ACTION ACT_Move:
{region "Primary"}
mcMoveAbsolute(	Axis					:= Axis,
				Execute					:= stMcAxisOnline.mcMoveAbsolute.bExecute,
				Position				:= stMcAxisOnline.mcMoveAbsolute.lrPosition,
				Velocity				:= stMcAxisOnline.mcMoveAbsolute.lrVelocity,
				Acceleration			:= stMcAxisOnline.mcMoveAbsolute.lrAcceleration,
				Deceleration			:= stMcAxisOnline.mcMoveAbsolute.lrDeceleration,
				Jerk					:= stMcAxisOnline.mcMoveAbsolute.lrJerk,
				BufferMode				:= stMcAxisOnline.mcMoveAbsolute.eBufferMode,
				Options					:= stMcAxisOnline.mcMoveAbsolute.stOptions,
				Done					=> stMcAxisOnline.mcMoveAbsolute.bDone,
				Busy					=> stMcAxisOnline.mcMoveAbsolute.bBusy,
				Active					=> stMcAxisOnline.mcMoveAbsolute.bActive,
				CommandAborted			=> stMcAxisOnline.mcMoveAbsolute.bCommandAborted,
				Error					=> stMcAxisOnline.mcMoveAbsolute.bError,
				ErrorID					=> stMcAxisOnline.mcMoveAbsolute.udiErrorID);

mcMoveRelative(	Axis					:= Axis,
				Execute					:= stMcAxisOnline.mcMoveRelative.bExecute,
				Distance				:= stMcAxisOnline.mcMoveRelative.lrDistance,
				Velocity				:= stMcAxisOnline.mcMoveRelative.lrVelocity,
				Acceleration			:= stMcAxisOnline.mcMoveRelative.lrAcceleration,
				Deceleration			:= stMcAxisOnline.mcMoveRelative.lrDeceleration,
				Jerk					:= stMcAxisOnline.mcMoveRelative.lrJerk,
				BufferMode				:= stMcAxisOnline.mcMoveRelative.eBufferMode,
				Options					:= stMcAxisOnline.mcMoveRelative.stOptions,
				Done					=> stMcAxisOnline.mcMoveRelative.bDone,
				Busy					=> stMcAxisOnline.mcMoveRelative.bBusy,
				Active					=> stMcAxisOnline.mcMoveRelative.bActive,
				CommandAborted			=> stMcAxisOnline.mcMoveRelative.bCommandAborted,
				Error					=> stMcAxisOnline.mcMoveRelative.bError,
				ErrorID					=> stMcAxisOnline.mcMoveRelative.udiErrorID);
				
mcMoveVelocity(	Axis					:= Axis,
				Execute					:= stMcAxisOnline.mcMoveVelocity.bExecute,
				Velocity				:= stMcAxisOnline.mcMoveVelocity.lrVelocity,
				Acceleration			:= stMcAxisOnline.mcMoveVelocity.lrAcceleration,
				Deceleration			:= stMcAxisOnline.mcMoveVelocity.lrDeceleration,
				Jerk					:= stMcAxisOnline.mcMoveVelocity.lrJerk,
				Direction				:= stMcAxisOnline.mcMoveVelocity.eDirection,
				BufferMode				:= stMcAxisOnline.mcMoveVelocity.eBufferMode,
				Options					:= stMcAxisOnline.mcMoveVelocity.stOptions,
				InVelocity				=> stMcAxisOnline.mcMoveVelocity.bInVelocity,
				Busy					=> stMcAxisOnline.mcMoveVelocity.bBusy,
				Active					=> stMcAxisOnline.mcMoveVelocity.bActive,
				CommandAborted			=> stMcAxisOnline.mcMoveVelocity.bCommandAborted,
				Error					=> stMcAxisOnline.mcMoveVelocity.bError,
				ErrorID					=> stMcAxisOnline.mcMoveVelocity.udiErrorID);
stMcAxisOnline.mcMoveVelocity.bDone		:= stMcAxisOnline.mcMoveVelocity.bInVelocity;

mcMoveModulo(	Axis					:= Axis,
				Execute					:= stMcAxisOnline.mcMoveModulo.bExecute,
				Position				:= stMcAxisOnline.mcMoveModulo.lrPosition,
				Velocity				:= stMcAxisOnline.mcMoveModulo.lrVelocity,
				Acceleration			:= stMcAxisOnline.mcMoveModulo.lrAcceleration,
				Deceleration			:= stMcAxisOnline.mcMoveModulo.lrDeceleration,
				Jerk					:= stMcAxisOnline.mcMoveModulo.lrJerk,
				Direction				:= stMcAxisOnline.mcMoveModulo.eDirection,
				BufferMode				:= stMcAxisOnline.mcMoveModulo.eBufferMode,
				Options					:= stMcAxisOnline.mcMoveModulo.stOptions,
				Done					=> stMcAxisOnline.mcMoveModulo.bDone,
				Busy					=> stMcAxisOnline.mcMoveModulo.bBusy,
				Active					=> stMcAxisOnline.mcMoveModulo.bActive,
				CommandAborted			=> stMcAxisOnline.mcMoveModulo.bCommandAborted,
				Error					=> stMcAxisOnline.mcMoveModulo.bError,
				ErrorID					=> stMcAxisOnline.mcMoveModulo.udiErrorID);
{endregion}
{region "Secondary"}
mcMoveAbsolute2(Axis					:= Axis,
				Execute					:= stMcAxisOnline.mcMoveAbsolute2.bExecute,
				Position				:= stMcAxisOnline.mcMoveAbsolute2.lrPosition,
				Velocity				:= stMcAxisOnline.mcMoveAbsolute2.lrVelocity,
				Acceleration			:= stMcAxisOnline.mcMoveAbsolute2.lrAcceleration,
				Deceleration			:= stMcAxisOnline.mcMoveAbsolute2.lrDeceleration,
				Jerk					:= stMcAxisOnline.mcMoveAbsolute2.lrJerk,
				BufferMode				:= stMcAxisOnline.mcMoveAbsolute2.eBufferMode,
				Options					:= stMcAxisOnline.mcMoveAbsolute2.stOptions,
				Done					=> stMcAxisOnline.mcMoveAbsolute2.bDone,
				Busy					=> stMcAxisOnline.mcMoveAbsolute2.bBusy,
				Active					=> stMcAxisOnline.mcMoveAbsolute2.bActive,
				CommandAborted			=> stMcAxisOnline.mcMoveAbsolute2.bCommandAborted,
				Error					=> stMcAxisOnline.mcMoveAbsolute2.bError,
				ErrorID					=> stMcAxisOnline.mcMoveAbsolute2.udiErrorID);

mcMoveRelative2(Axis					:= Axis,
				Execute					:= stMcAxisOnline.mcMoveRelative2.bExecute,
				Distance				:= stMcAxisOnline.mcMoveRelative2.lrDistance,
				Velocity				:= stMcAxisOnline.mcMoveRelative2.lrVelocity,
				Acceleration			:= stMcAxisOnline.mcMoveRelative2.lrAcceleration,
				Deceleration			:= stMcAxisOnline.mcMoveRelative2.lrDeceleration,
				Jerk					:= stMcAxisOnline.mcMoveRelative2.lrJerk,
				BufferMode				:= stMcAxisOnline.mcMoveRelative2.eBufferMode,
				Options					:= stMcAxisOnline.mcMoveRelative2.stOptions,
				Done					=> stMcAxisOnline.mcMoveRelative2.bDone,
				Busy					=> stMcAxisOnline.mcMoveRelative2.bBusy,
				Active					=> stMcAxisOnline.mcMoveRelative2.bActive,
				CommandAborted			=> stMcAxisOnline.mcMoveRelative2.bCommandAborted,
				Error					=> stMcAxisOnline.mcMoveRelative2.bError,
				ErrorID					=> stMcAxisOnline.mcMoveRelative2.udiErrorID);
				
mcMoveVelocity2(Axis					:= Axis,
				Execute					:= stMcAxisOnline.mcMoveVelocity2.bExecute,
				Velocity				:= stMcAxisOnline.mcMoveVelocity2.lrVelocity,
				Acceleration			:= stMcAxisOnline.mcMoveVelocity2.lrAcceleration,
				Deceleration			:= stMcAxisOnline.mcMoveVelocity2.lrDeceleration,
				Jerk					:= stMcAxisOnline.mcMoveVelocity2.lrJerk,
				Direction				:= stMcAxisOnline.mcMoveVelocity2.eDirection,
				BufferMode				:= stMcAxisOnline.mcMoveVelocity2.eBufferMode,
				Options					:= stMcAxisOnline.mcMoveVelocity2.stOptions,
				InVelocity				=> stMcAxisOnline.mcMoveVelocity2.bInVelocity,
				Busy					=> stMcAxisOnline.mcMoveVelocity2.bBusy,
				Active					=> stMcAxisOnline.mcMoveVelocity2.bActive,
				CommandAborted			=> stMcAxisOnline.mcMoveVelocity2.bCommandAborted,
				Error					=> stMcAxisOnline.mcMoveVelocity2.bError,
				ErrorID					=> stMcAxisOnline.mcMoveVelocity2.udiErrorID);
stMcAxisOnline.mcMoveVelocity2.bDone	:= stMcAxisOnline.mcMoveVelocity2.bInVelocity;

mcMoveModulo2(	Axis					:= Axis,
				Execute					:= stMcAxisOnline.mcMoveModulo2.bExecute,
				Position				:= stMcAxisOnline.mcMoveModulo2.lrPosition,
				Velocity				:= stMcAxisOnline.mcMoveModulo2.lrVelocity,
				Acceleration			:= stMcAxisOnline.mcMoveModulo2.lrAcceleration,
				Deceleration			:= stMcAxisOnline.mcMoveModulo2.lrDeceleration,
				Jerk					:= stMcAxisOnline.mcMoveModulo2.lrJerk,
				Direction				:= stMcAxisOnline.mcMoveModulo2.eDirection,
				BufferMode				:= stMcAxisOnline.mcMoveModulo2.eBufferMode,
				Options					:= stMcAxisOnline.mcMoveModulo2.stOptions,
				Done					=> stMcAxisOnline.mcMoveModulo2.bDone,
				Busy					=> stMcAxisOnline.mcMoveModulo2.bBusy,
				Active					=> stMcAxisOnline.mcMoveModulo2.bActive,
				CommandAborted			=> stMcAxisOnline.mcMoveModulo2.bCommandAborted,
				Error					=> stMcAxisOnline.mcMoveModulo2.bError,
				ErrorID					=> stMcAxisOnline.mcMoveModulo2.udiErrorID);
{endregion}
END_ACTION

ACTION ACT_Power:
mcPower(	Axis						:= Axis,									//
			Enable						:= stMcAxisOnline.mcPower.bEnable,
			Enable_Positive				:= stMcAxisOnline.mcPower.bEnable_Positive,
			Enable_Negative				:= stMcAxisOnline.mcPower.bEnable_Negative,
			Override					:= stMcAxisOnline.mcPower.lrOverride,
			BufferMode					:= stMcAxisOnline.mcPower.eBufferMode,
			Options						:= stMcAxisOnline.mcPower.stOptions,
			Status						=> stMcAxisOnline.mcPower.bStatus,
			Busy						=> stMcAxisOnline.mcPower.bBusy,
			Active						=> stMcAxisOnline.mcPower.bActive,
			Error						=> stMcAxisOnline.mcPower.bError,
			ErrorID						=> stMcAxisOnline.mcPower.udiErrorID);
END_ACTION

ACTION ACT_ResetAndDiag:
tonGetDriveDiag(IN:= stMcAxisOnline.stError.bDriveError AND NOT tonGetDriveDiag.Q, PT:= T#5S, Q=> , ET=> );

IF Axis.Status.OpMode.SimulationAxis THEN
	mcReset(
		Axis						:= Axis,
		Execute						:= stMcAxisOnline.mcReset.bExecute,
		Done						=> stMcAxisOnline.mcReset.bDone,
		Busy						=> stMcAxisOnline.mcReset.bBusy,
		Error						=> stMcAxisOnline.mcReset.bError,
		ErrorID						=> stMcAxisOnline.mcReset.udiErrorID);	
ELSE
	fbReadChannelErrorCode(
		Reset:=					stMcAxisOnline.mcReset.bExecute,
		GetDiag				:=	(stMcAxisOnline.stChannelErrorCode.bExecute OR tonGetDriveDiag.Q),
		Axis				:=	Axis , 
		stAX5000Diag		:=	stAX5000Diag , 
		Error				=> 	stMcAxisOnline.mcReset.bError , 
		AdsErrId			=>	stMcAxisOnline.mcReset.udiErrorID , 
		SercosErrId			=>	stMcAxisOnline.stChannelErrorCode.uiAdsErrId, //???
		ResetAct			=> , 
		DiagAct				=> , 
		Busy				=> 	stMcAxisOnline.mcReset.bBusy );
	
	stMcAxisOnline.stChannelErrorCode.bError 				:= stAX5000Diag.bC1DError;
	stMcAxisOnline.stChannelErrorCode.uiChannelErrorCode 	:= UDINT_TO_UINT (stAX5000Diag.iDiagNumber);
	stMcAxisOnline.stChannelErrorCode.uiChannelErrorCodeHex := UDINT_TO_UINT (stAX5000Diag.iDiagNumber);
END_IF
END_ACTION

ACTION ACT_SetPosition:
mcSetPosition(		Axis				:= Axis,
					Execute				:= stMcAxisOnline.mcSetPosition.bExecute,
					Position			:= stMcAxisOnline.mcSetPosition.lrPosition,
					Mode				:= stMcAxisOnline.mcSetPosition.bMode,
					Options				:= stMcAxisOnline.mcSetPosition.stOptions,
					Done				=> stMcAxisOnline.mcSetPosition.bDone,
					Busy				=> stMcAxisOnline.mcSetPosition.bBusy,
					Error				=> stMcAxisOnline.mcSetPosition.bError,
					ErrorID				=> stMcAxisOnline.mcSetPosition.udiErrorID);
END_ACTION

ACTION ACT_SetPositionIO:
fbSetPositionOffset(
	bExecute			:= stMcAxisOnline.stSetPositionOffset.bExecute , 
	lrPosition			:= stMcAxisOnline.stSetPositionOffset.lrPosition , 
	bRelative			:= stMcAxisOnline.stSetPositionOffset.bRelative , 
	eFeedback			:= stMcAxisOnline.stSetPositionOffset.eFeedback , 
	eMemory				:= stMcAxisOnline.stSetPositionOffset.eMemory , 
	bBusy				=> stMcAxisOnline.stSetPositionOffset.bBusy , 
	bError				=> stMcAxisOnline.stSetPositionOffset.bError, 
	udiErrorID			=> stMcAxisOnline.stSetPositionOffset.udiErrorID, 
	uiSoEErrorID		=> stMcAxisOnline.stSetPositionOffset.uiSecErrId,
	Axis				:= Axis );
END_ACTION

ACTION ACT_States:
// Read States and forward main states
Axis.ReadStatus();
stMcAxisOnline.stStatus.stAxisStatus		:= Axis.Status;
stMcAxisOnline.stStatus.dwAxisId			:= Axis.NcToPlc.AxisId;
stMcAxisOnline.stStatus.bNcError			:= Axis.Status.Error;
stMcAxisOnline.stStatus.udiNcErrorCode		:= Axis.Status.ErrorID;
stMcAxisOnline.stStatus.udiNcErrorCodeHex	:= Axis.Status.ErrorID;

stMcAxisOnline.stStatus.sAxisName			:= stMcAxisOnline.stAxisParameter.sAxisName;
stMcAxisOnline.stStatus.lrActPos			:= Axis.NcToPlc.ActPos;
stMcAxisOnline.stStatus.lrModuloActPos		:= Axis.NcToPlc.ModuloActPos;
stMcAxisOnline.stStatus.lrActVelo			:= Axis.NcToPlc.ActVelo;
stMcAxisOnline.stStatus.lrActAcc			:= Axis.NcToPlc.ActAcc;
stMcAxisOnline.stStatus.lrActTorque			:= Axis.NcToPlc.ActTorque;
stMcAxisOnline.stStatus.lrPosDiff			:= Axis.NcToPlc.PosDiff;
stMcAxisOnline.stStatus.lrSetPos			:= Axis.NcToPlc.SetPos;
stMcAxisOnline.stStatus.lrSetVelo			:= Axis.NcToPlc.SetVelo;
stMcAxisOnline.stStatus.lrSetAcc			:= Axis.NcToPlc.SetAcc;
stMcAxisOnline.stStatus.lrSetTorque			:= Axis.NcToPlc.SetTorque;
stMcAxisOnline.stStatus.lrPosDiff			:= Axis.NcToPlc.PosDiff;
stMcAxisOnline.stStatus.bAxisReady			:= Axis.Status.Operational;
stMcAxisOnline.stStatus.bHomed				:= Axis.Status.Homed;
stMcAxisOnline.stStatus.bCoupled			:= Axis.Status.Coupled;

// zezwolenie na zjazd z krancowki hw
Axis.PlcToNc.ControlDWord.8				:= stMcAxisOnline.stStatus.bAcceptBlockedDrive;
END_ACTION

ACTION ACT_Stop:
mcHalt(		Axis						:= Axis,
			Execute						:= stMcAxisOnline.mcHalt.bExecute,
			Deceleration				:= stMcAxisOnline.mcHalt.lrDeceleration,
			Jerk						:= stMcAxisOnline.mcHalt.lrJerk,
			BufferMode					:= stMcAxisOnline.mcHalt.eBufferMode,
			Options						:= stMcAxisOnline.mcHalt.stOptions,
			Done						=> stMcAxisOnline.mcHalt.bDone,
			Busy						=> stMcAxisOnline.mcHalt.bBusy,
			Active						=> stMcAxisOnline.mcHalt.bActive,
			CommandAborted				=> stMcAxisOnline.mcHalt.bCommandAborted,
			Error						=> stMcAxisOnline.mcHalt.bError,
			ErrorID						=> stMcAxisOnline.mcHalt.udiErrorID);
			
mcStop(		Axis						:= Axis,
			Execute						:= stMcAxisOnline.mcStop.bExecute,
			Deceleration				:= stMcAxisOnline.mcStop.lrDeceleration,
			Jerk						:= stMcAxisOnline.mcStop.lrJerk,
			Options						:= stMcAxisOnline.mcStop.stOptions,
			Done						=> stMcAxisOnline.mcStop.bDone,
			Busy						=> stMcAxisOnline.mcStop.bBusy,
			Active						=> stMcAxisOnline.mcStop.bActive,
			CommandAborted				=> stMcAxisOnline.mcStop.bCommandAborted,
			Error						=> stMcAxisOnline.mcStop.bError,
			ErrorID						=> stMcAxisOnline.mcStop.udiErrorID);
			
mcStopSS2(	Axis						:= Axis,
			Execute						:= stMcAxisOnline.mcSS2.bExecute,
			Deceleration				:= stMcAxisOnline.mcSS2.lrDeceleration,
			Jerk						:= stMcAxisOnline.mcSS2.lrJerk,
			Options						:= stMcAxisOnline.mcSS2.stOptions,
			Done						=> stMcAxisOnline.mcSS2.bDone,
			Busy						=> stMcAxisOnline.mcSS2.bBusy,
			Active						=> stMcAxisOnline.mcSS2.bActive,
			CommandAborted				=> stMcAxisOnline.mcSS2.bCommandAborted,
			Error						=> stMcAxisOnline.mcSS2.bError,
			ErrorID						=> stMcAxisOnline.mcSS2.udiErrorID);
			
mcStopSS1(	Axis						:= Axis,
			Execute						:= stMcAxisOnline.mcSS1.bExecute,
			Deceleration				:= stMcAxisOnline.mcSS1.lrDeceleration,
			Jerk						:= stMcAxisOnline.mcSS1.lrJerk,
			Options						:= stMcAxisOnline.mcSS1.stOptions,
			Done						=> stMcAxisOnline.mcSS1.bDone,
			Busy						=> stMcAxisOnline.mcSS1.bBusy,
			Active						=> stMcAxisOnline.mcSS1.bActive,
			CommandAborted				=> stMcAxisOnline.mcSS1.bCommandAborted,
			Error						=> stMcAxisOnline.mcSS1.bError,
			ErrorID						=> stMcAxisOnline.mcSS1.udiErrorID);
// SS1 - after MC_Stop function we have to disable drive			
stMcAxisOnline.mcPower.bEnable R= stMcAxisOnline.mcPower.bEnable_Positive R= stMcAxisOnline.mcPower.bEnable_Negative R= (stMcAxisOnline.mcSS1.bDone OR stMcAxisOnline.mcSS1.bCommandAborted OR stMcAxisOnline.mcSS1.bError);
END_ACTION

ACTION ACT_SWLimitSwitch:
fbNcLimitSwitch(	udiAxisID		:= Axis.NcToPlc.AxisId, 
					bRead			:= stMcAxisOnline.stNcLimitSwitch.bRead, 
					bWrite			:= stMcAxisOnline.stNcLimitSwitch.bWrite, 
					bReset			:= stMcAxisOnline.stNcLimitSwitch.bReset, 
					lrSetMinPos		:= stMcAxisOnline.stNcLimitSwitch.lrSetMinPos, 
					lrSetMaxPos		:= stMcAxisOnline.stNcLimitSwitch.lrSetMaxPos, 
					bSetMinMon		:= stMcAxisOnline.stNcLimitSwitch.bSetMinMon, 
					bSetMaxMon		:= stMcAxisOnline.stNcLimitSwitch.bSetMaxMon, 
					bBusy			=> stMcAxisOnline.stNcLimitSwitch.bBusy, 
					bError			=> stMcAxisOnline.stNcLimitSwitch.bError, 
					udiErrorID		=> stMcAxisOnline.stNcLimitSwitch.udiErrorID, 
					lrActMinPos		=> stMcAxisOnline.stNcLimitSwitch.lrActMinPos, 
					lrActMaxPos		=> stMcAxisOnline.stNcLimitSwitch.lrActMaxPos, 
					bActMinMon		=> stMcAxisOnline.stNcLimitSwitch.bActMinMon, 
					bActMaxMon		=> stMcAxisOnline.stNcLimitSwitch.bActMaxMon);
END_ACTION

END_FUNCTION_BLOCK

// ---- POUs/FB/POUsAxisOnline/AX5000/FB_SetPositionOffset.TcPOU
//==================================================================================================
//							Beckhoff Automation Poland
//									07.06.2018
//	Blok do uzupełniania offsetu w enkoderze/AX5000
//	Obsluguje bledy zwiazane z wymiana silnika na nowy - bez wpisanego offsetu.
//	Naprawia błąd: 	0x0000F340- Position offset invalid.
//					0x0000F341- Position offset: No position offset excisting.
//	Aby wpisać wartość, silnik musi być wyłączony.
//	Niezbędne biblioteki:
//	Tc2_MC2;	Tc2_Utilities;	Tc2_MC2_Drive;	Tc2_EtherCAT, Tc2_Drive;
//
//	v2.4 || TC v 3.1.4022.20 || - Usuniecie nieużywanych zmiennych, zabezpieczenie przed zerowa pozycja, optymalizacje
//	v2.2 || TC v 3.1.4022.2	 || - Poprawka w komentarzu, uiSoEErrorID zamiast udiSoEErrorID
//	v2.1 || TC v 3.1.4022.0	 || - Uproszczono kod
//	v2.0 || TC v 3.1.4022.0	 || - Dodano obsługę AX52xx, przebudowano bloczek z wykorzystaniem FB_ChangeSlaveState
//	v1.0 || TC v 3.1.4020.32 || - Pierwsza wersja
//==================================================================================================
FUNCTION_BLOCK FB_SetPositionOffset
VAR_INPUT
	bExecute								: BOOL;							// rising edge starts sequence
	lrPosition								: LREAL		:=	0.001;			// Write new encoder position
	bRelative								: BOOL;							// When this flag is set, the position is relatively interpreted
	eFeedback								: E_PositionOffsetFeedback;		// ePositionOffsetFeedback1:= 0			ePositionOffsetFeedback2 := 1
	eMemory									: E_PositionOffsetMemory;		// ePositionOffsetMemory_Encoder:= 0	ePositionOffsetMemory_Drive := 1
END_VAR
VAR_OUTPUT
	bBusy									: BOOL;
	bError									: BOOL;	
	udiErrorID								: UDINT;						// bError=TRUE AND udiErrorID=0 means state request timeout
	uiSoEErrorID							: UINT;
	udiADSerrorID							: UDINT;
END_VAR
VAR_IN_OUT
	Axis									: AXIS_REF;
END_VAR
VAR CONSTANT
	NCIDXG_AXPARMS							: UDINT			:= 16#4000;		// ADS group number to axis parameters 
	NCIDXO_AXP_HWAMSADDR					: UDINT			:= 16#31;		// ADS offset to drive channel
END_VAR
VAR
	rtExecute								: R_TRIG;						// bExecute triggers start
	fbSoEReset								: FB_SoEReset;
	fbSoEWritePassword						: FB_SoEWritePassword;			// unlock P-0-0278
	fbSoEAX5000SetPositionOffset			: FB_SoEAX5000SetPositionOffset;
	fbSoEReadDiagNumber						: FB_SoEReadDiagNumber;	
	fbSoEWrite_ByDriveRef					: FB_SoEWrite_ByDriveRef;
	fbSoERead_ByDriveRef					: FB_SoERead_ByDriveRef;
	fbChangeSlaveState						: FB_ChangeEtherCATSlaveState;
	fbAdsRead								: ADSREAD;
	stPlcDriveRef							: ST_PlcDriveRef;				// ADS buffer (need to change aNetId into sNetId)
	stDriveRef								: ST_DriveRef;					// come from stPlcDriveRef
	bDualChannel							: BOOL;
	stSoE_String							: ST_SoE_String;				// buffer for byDualChannel
	P_0_0278_Value							: WORD;							//	0- NO	1- YES
	iStep									: INT;							// Actual Step
	iLastStep								: INT;							// Last step before error
END_VAR

rtExecute	(CLK:= bExecute );

CASE iStep	OF

	0:																//	Enable FB, lock input parameters
		IF rtExecute.Q THEN
			bBusy							:= TRUE;
			bError							:= FALSE;
			udiErrorID						:= 0;
			uiSoEErrorID					:= 0;
			udiADSerrorID					:= 0;
			iLastStep						:= 0;
			IF ABS(lrPosition) < LREAL#0.0001 THEN
				fbSoEAX5000SetPositionOffset.Position := LREAL#0.0001;
			ELSE
				fbSoEAX5000SetPositionOffset.Position := lrPosition; 
			END_IF
			fbSoEAX5000SetPositionOffset.Memory	:= eMemory;
			fbSoEAX5000SetPositionOffset.Relative := bRelative;
			fbSoEAX5000SetPositionOffset.Feedback := eFeedback;
			iStep							:= iStep+10;
		END_IF			

	10:																// Get Drive channel from AXIS_REF by ADS
		fbAdsRead.NETID						:= '';
		fbAdsRead.PORT						:= AMSPORT_R0_NC;		// set ADS Port to NC
		fbAdsRead.IDXGRP					:= NCIDXG_AXPARMS + Axis.NcToPlc.AxisId;	// set ADS Group to AXIS Parameters
		fbAdsRead.IDXOFFS					:= NCIDXO_AXP_HWAMSADDR;// set ADS offset to channel number
		fbAdsRead.LEN						:= SIZEOF(stPlcDriveRef);
		fbAdsRead.DESTADDR					:= ADR(stPlcDriveRef);
		fbAdsRead.TMOUT						:= T#5S;
		fbAdsRead.READ						:= TRUE;
		iStep								:= istep+10;
		
	20:																// reading actual channel (DriveNo) from AXIS_REF	
		fbAdsRead.READ						:= FALSE;
		IF NOT fbAdsRead.BUSY THEN
			IF  NOT fbAdsRead.ERR THEN
				iStep							:= iStep+10;	
				stDriveRef.sNetId				:= F_CreateAmsNetId(stPlcDriveRef.aNetId);	// change AmsNetId array into string
				stDriveRef.nSlaveAddr			:= stPlcDriveRef.nSlaveAddr;
				stDriveRef.nDriveNo				:= stPlcDriveRef.nDriveNo;	
				fbChangeSlaveState.sEtherCAT_NetID:= stDriveRef.sNetId;
				fbChangeSlaveState.nSlaveAddr	:= stDriveRef.nSlaveAddr;
			ELSIF fbAdsRead.ERR THEN
				udiADSerrorID					:= fbAdsRead.ERRID;
				iLastStep						:= iStep;
				iStep							:= 999;				
			END_IF
		END_IF
		
	30:																// Read drive diag number
		fbSoEReadDiagNumber.NetId			:= '';
		fbSoEReadDiagNumber.Execute			:= TRUE;
		iStep								:= iStep+10;

	40:																// Choose method
		fbSoEReadDiagNumber.Execute			:= FALSE;
		IF NOT fbSoEReadDiagNumber.Busy THEN
			IF fbSoEReadDiagNumber.DiagNumber = (16#F341 OR 16#F340) THEN
				iStep						:= 50;					// Position errors -> Reset errors and write 
			ELSIF	fbSoEReadDiagNumber.DiagNumber >= (16#F000) THEN
				iLastStep					:= iStep;				// Do nothing in other error states
				iStep						:= 999;
			ELSE												
				iStep						:= 200;					// Drive Ready -> Write without changing OP State			
			END_IF
		END_IF
	
	50:																// Request INIT State
		fbChangeSlaveState.byReguestedState	:= EC_DEVICE_STATE_INIT;
		fbChangeSlaveState.bExecute			:= TRUE;
		iStep								:= iStep+10;

	60,80:															// Wait till state changed
		fbChangeSlaveState.bExecute			:= FALSE;
		IF NOT fbChangeSlaveState.bBusy THEN
			IF NOT fbChangeSlaveState.bError THEN
				iStep							:= iStep+10;
			ELSE
				udiErrorID						:= fbChangeSlaveState.udiErrorID;
				iLastStep						:= iStep;
				iStep 							:= 999;
			END_IF
		END_IF
		
	70:																// Request PreOP State	
		fbChangeSlaveState.byReguestedState	:= EC_DEVICE_STATE_PREOP;
		fbChangeSlaveState.bExecute			:= TRUE;
		iStep								:= iStep+10;
		
	90:																// Write drive password (unlock P-0-0278)
		fbSoEWritePassword.Password.strData	:= 'AX5000';
		fbSoEWritePassword.NetId			:= '';
		fbSoEWritePassword.Execute			:= TRUE;
		iStep								:= iStep + 10;
		
	100:															// wait till password passes
		fbSoEWritePassword.Execute			:= FALSE;
		IF NOT fbSoEWritePassword.Busy THEN
			IF NOT fbSoEWritePassword.Error THEN
				iStep							:= iStep + 10;
			ELSE 
				udiADSerrorID					:= fbSoEWritePassword.AdsErrId;
				uiSoEErrorID					:= fbSoEWritePassword.SercosErrId;
				iLastStep						:= iStep;
				iStep							:= 999;
			END_IF
		END_IF
		
	110:															// Ignore offset error (P-0-0278), channel 1	
		P_0_0278_Value						:= 1;
		fbSoEWrite_ByDriveRef.stDriveRef	:= stDriveRef;
		fbSoEWrite_ByDriveRef.stDriveRef.nDriveNo:= 0;
		fbSoEWrite_ByDriveRef.nIdn			:= P_0_IDN  + 278;		// SoE Parameters Group P-0-IDN offset
		fbSoEWrite_ByDriveRef.nElement		:= EC_SOE_ELEMENT_VALUE;// Change value of the parameter
		fbSoEWrite_ByDriveRef.pSrcBuf		:= ADR(P_0_0278_Value);
		fbSoEWrite_ByDriveRef.cbBufLen		:= SIZEOF(P_0_0278_Value);
		fbSoEWrite_ByDriveRef.bExecute		:= TRUE;
		iStep								:= iStep + 10;				
		
	120,160:														// Writing done ?		
		fbSoEWrite_ByDriveRef.bExecute		:= FALSE;
		IF NOT fbSoEWrite_ByDriveRef.bBusy THEN
			IF NOT fbSoEWrite_ByDriveRef.bError THEN
				iStep							:= iStep + 10;
			ELSE
				udiADSerrorID					:= fbSoEWrite_ByDriveRef.iAdsErrId;
				uiSoEErrorID					:= fbSoEWrite_ByDriveRef.iSercosErrId;
				iLastStep						:= iStep;
				iStep							:= 999;
			END_IF	
		END_IF
		
	130:															// reset second channel if needed
		fbSoERead_ByDriveRef.stDriveRef		:= stDriveRef;
		fbSoERead_ByDriveRef.nIdn			:= P_0_IDN  + 324;		// SoE Parameters Group P-0-IDN offset
		fbSoERead_ByDriveRef.nElement		:= EC_SOE_ELEMENT_VALUE;// Change value of the parameter
		fbSoERead_ByDriveRef.pDstBuf		:= ADR(stSoE_String);
		fbSoERead_ByDriveRef.cbBufLen		:= SIZEOF(stSoE_String);
		fbSoERead_ByDriveRef.bExecute		:= TRUE;
		iStep								:= iStep + 10;				
		
	140:															// Reading done ?	skip reseting channel 2 for AX51xx	
		fbSoERead_ByDriveRef.bExecute		:= FALSE;
		IF NOT fbSoERead_ByDriveRef.bBusy THEN
			IF NOT fbSoERead_ByDriveRef.bError THEN
				bDualChannel := STRING_TO_BYTE(MID(stSoE_String.strData, 1, 4)) = 2;		// Sprawdza nazwe AX5xxx i rozpoznaje ilosc kanalow
				IF bDualChannel THEN
					iStep						:= iStep + 10;			// reset channel 2
				ELSE
					iStep						:= iStep + 30;			// skip reseting channel 2
				END_IF
			ELSE
				udiADSerrorID					:= fbSoERead_ByDriveRef.iAdsErrId;
				uiSoEErrorID					:= fbSoERead_ByDriveRef.iSercosErrId;
				iLastStep						:= iStep;
				iStep							:= 999;
			END_IF	
		END_IF
		
	150:															// Ignore offset error (P-0-0278), channel 2
		fbSoEWrite_ByDriveRef.stDriveRef.nDriveNo:= 1;
		fbSoEWrite_ByDriveRef.bExecute		:= TRUE;
		iStep								:= iStep + 10;

	170:															// Reset Drive (S-0-0099)
		fbSoEReset.Execute					:= TRUE; 
		fbSoEReset.NetId					:= ''; 
		iStep								:= iStep + 10;
		
	180:															// Wait for drive reset (S-0-0099)
		fbSoEReset.Execute					:= FALSE;
		IF NOT fbSoEReset.Busy THEN
			IF NOT fbSoEReset.Error THEN
				iStep							:= iStep + 10;
			ELSE
				udiADSerrorID					:= fbSoEReset.AdsErrId;
				uiSoEErrorID					:= fbSoEReset.SercosErrId;
				iLastStep						:= iStep;
				iStep							:= 999;
			END_IF
		END_IF
		
	190:															// Request OP State
		fbChangeSlaveState.byReguestedState	:= EC_DEVICE_STATE_OP;
		fbChangeSlaveState.bExecute			:= TRUE;
		iStep								:= iStep+10;
	
	200:															// Wait till state changed
		fbChangeSlaveState.bExecute			:= FALSE;	
		IF NOT fbChangeSlaveState.bBusy THEN
			IF NOT fbChangeSlaveState.bError THEN
				iStep							:= iStep+10;
			ELSE
				udiErrorID						:= fbChangeSlaveState.udiErrorID;
				iLastStep						:= iStep;
				iStep 							:= 999;
			END_IF				
		END_IF
		
	210:															// Set new encoder offset	
		fbSoEAX5000SetPositionOffset.Feedback:= ePositionOffsetFeedback1;	// set to feedback 1 only
		fbSoEAX5000SetPositionOffset.Execute:= TRUE; 
		iStep								:= iStep + 10;

	220:															//	offset set already?
		fbSoEAX5000SetPositionOffset.Execute:= FALSE;
		IF NOT fbSoEAX5000SetPositionOffset.Busy THEN
			IF NOT fbSoEAX5000SetPositionOffset.Error THEN
				iStep							:= iStep + 10;
			ELSE
				udiErrorID						:= fbSoEAX5000SetPositionOffset.ErrorID;
				iLastStep						:= iStep;
				iStep							:= 999;
			END_IF
		END_IF
	
	230:															//	FB Termination
		bBusy								:= FALSE;
		iStep								:= 0;

	999:															//	ERROR State
		bBusy								:=	FALSE;
		bError								:=	TRUE;
		iStep								:=	0;
	
END_CASE

fbAdsRead();
fbChangeSlaveState();
fbSoEWritePassword(Axis:=Axis);
fbSoEAX5000SetPositionOffset(Axis:=Axis);
fbSoEReadDiagNumber(Axis:=Axis);
fbSoEReset(Axis:=Axis);
fbSoEWrite_ByDriveRef();
fbSoERead_ByDriveRef();

END_FUNCTION_BLOCK

// ---- POUs/FB/POUsAxisOnline/AX5000/FB_MotorMonitoringAX5000.TcPOU
//==================================================================================================
//							Beckhoff Automation Poland
//									22.09.2020
//	Blok funkcyjny pozwala na monitorowanie i ograniczanie momentu oraz monitoring parametru I2T dla AX5xxx.
//	Zmienne do zlinkowania zadeklarowane są wewnątrz bloku.
//	Ograniczenie i monitorowanie momentu
//	Ograniczenie momentu podawane jest przez wejście rTorqueLimit.
//	Na wyjściu podana jest wartość surowa w %, jak i przeskalowana na A (prąd) i Nm (moment).
//	Blok zwraca wartości bieżące, przefiltrowane i maksymalne.
//	Wartości maksymalne mogą być wyzerowane za pomocą zmiennej bReset.
//	Wewnętrznie wykorzystany jest blok FB_FilterEx.
//	I2T: 	Określamy okno czasowe pomiaru
//	Biblioteki: Tc2_MC2, Tc2_MC2_Drive, Tc2_Drive, Tc2_EtherCAT
//
// 	v1.4	|| TC v 3.1.4024.10		|| dostosowany do FW 2.13
// 	v1.3	|| TC v 3.1.4022.22		|| optymalizacja kod poprawiony blad wyliczenia Torque filtered
// 	v1.2	|| TC v 3.1.4022.22		|| optymalizacja kodu
// 	v1.1	|| TC v 3.1.4022.16		|| optymalizacja kodu, poprawiona flaga initialized
//  v1.0	|| TC v 3.1.4022.16		|| bazuje na FB_TorqueMonitoringEx2, dodane wyjscia zgodne z blokiem do AX8000 
//==================================================================================================
FUNCTION_BLOCK FB_MotorMonitoringAX5000
VAR CONSTANT
	rTorqueLimitLow					: REAL 		:= 0.01;				// Low limit used for bipolar torque limit value
	rTorqueLimitHigh				: REAL		:= 100.0;				// High limit used for bipolar torque limit value
END_VAR
VAR_INPUT
	bReset							: BOOL;
	rTorqueLimit					: REAL 		:= rTorqueLimitHigh; 	// Bipolar torque limit: 0-500%, resolution 0.1%, value goes to: 16#6072 (Ch A)/ 16#6872 (Ch B)
	tI2T_Window						: TIME 		:= T#100S;				// Has to be Task time * 100 * x 
																		// x - how many probes per measurement
																		// Samples - Task: 2 ms - tI2T_Window min 200 ms (1 probe), 100 probes then 20 s
																		// Task: 10 ms - tI2T_Window min 1 s (1 probe), 100 probes then 100 s
																		// If not proper time entered then it'll be adjusted
END_VAR
VAR_OUTPUT
	bError							: BOOL; 							// Communication error
	uiAdsErrId						: UINT;								// Forwarded output FB_SoeRead
	uiSercosErrId					: UINT;								// Forwarded output FB_SoeRead
	bInitialized					: BOOL;								// TRUE - Motor data read without errors, so it's possible to calculate torqe and current values in metric units
	bWarning						: BOOL;								// Overcurrent (rCurrentF > rRatedCurrent)
	rWarningCurrent					: REAL; 							// P_0_0093_Value in [A]
	rTorquePerc						: REAL;								// [%]
	rTorquePercMax					: REAL;								// Max [%]	
	rTorque							: REAL; 							// [Nm]
	rTorqueF						: REAL;								// Filtered
	rTorqueMax						: REAL;								// Max
	rCurrent						: REAL; 							// [A]
	rCurrentF						: REAL;								// Filtered
	rCurrentMax						: REAL;								// Max
	rI2T							: REAL; 							// % nominal
	rI2TMax							: REAL;
END_VAR
VAR_IN_OUT
	Axis							: AXIS_REF;
END_VAR
VAR
//======================== Internal =============================
	rTorqueRAW						: REAL; 							// -1000 .. 1000 - RAW values the same as process image	
	rContinuousStallTorque			: REAL; 							// P_0_0070_Value [Nm]
	rContinuousStallCurrent			: REAL; 							// S_0_0111_Value [A]
	rPeakCurrent					: REAL; 							// P_0_0092_Value in [A]
	rSfTorque						: REAL; 							// A --> Nm P_0_0070_Value/S_0_0111_Value [Nm/A]
	rSfCurrent						: REAL; 							// RAW --> A (-1000..1000 --> - rPeakCurrent .. rPeakCurrent)
	bFirstCycle						: BOOL := TRUE;
	iFW_High						: INT;
	iFW_Low							: INT;
	bDriveFirmware_GE_2_10			: BOOL;								// From FW >= 2.10 - different image size
	iFWPos							: INT;
	iFWLen							: INT;
	sDriveFW						: STRING(66);
	uiBipolarTorqueLimitValue AT %Q*	: UINT; 						// Raw data, linked to Bipolar torque limit value MDT, S-0-0092
	iStep							: INT;
	wInitErrorCount					: WORD;								// Initialization error counter, if bigger then 10 then error
	arr_S_0_0030_Value				: ARRAY [1..66] OF BYTE;			// till FW 2.10 total len is 66 bytes (2 - Act len, 2 - Max len, 62 - String 
	S_0_0030_Value					: STRING(61);
	P_0_0092_Value					: DWORD;
	P_0_0093_Value					: DWORD;
	P_0_0070_Value					: DWORD;
	S_0_0111_Value					: DWORD;
//========================== I2T ================================
	bCalculateI2T					: BOOL;								// TRUE in cycle when recalculation I2T necessary
	bBufferFull						: BOOL;								// TRUE when array buffer is full
	BIndex							: BYTE;								// Task no
	tI2T_WindowOld					: TIME;								// Old time window to reinit I2T calculation if necessary
	wProbeCyclesCount				: WORD;								// No of cycles for one I2T probe
	wCyclesCount					: WORD;								// Act no of cycles for one I2T probe
	wNoOfCycles						: WORD;								// Total cycles count for I2T window
	wNoOfProbes						: WORD;								// Actual number of probes for I2T calculation
	i								: INT;								// FOR loop
	rCycleTime						: REAL;								// Task time in [ms]
	rI2T_Window						: REAL;								// Time window in [ms]
	rCurrentPom						: REAL;								// Sum of current values in probe
	rCurrentAverage					: REAL;								// Arithmetical average
	rI2T_Nominal					: REAL;								// I2T for In
	rI2T_Actual						: REAL;								// I2T for real values
	arrI2TBuffer					: ARRAY[1..100] OF REAL;			// Buffer window to calculate I2T
//========================== FBs ================================
	rtReset							: R_TRIG;							// Reset trigger
	tonWait							: TON;								// Wait timer
	fbFilterEx						: FB_FilterEx;						// Filter
	fbSoERead						: FB_SoeRead;						// FB for read SoE parameters
	fbGETCURTASKINDEX   			: GETCURTASKINDEX;					// FB to check task no
//===============================================================
END_VAR

//===== Initialization, reinitialization and reset  =============
ACT_Init_Reset();
//=================== Call triggers and timers ==================
tonWait(IN:= NOT tonWait.Q, PT:= T#1S);
//============= Read params and calculations ====================
CASE iStep OF

	0: 	// Read S_0_0030 - Manufacturer version

		fbSoERead.Idn 					:= S_0_IDN + 30;
		fbSoERead.Element				:= EC_SOE_ELEMENT_VALUE;
		fbSoERead.pDstBuf				:= ADR(arr_S_0_0030_Value);
		fbSoERead.BufLen				:= SIZEOF(arr_S_0_0030_Value);
		fbSoERead.Execute				:= TRUE;
		iStep 							:= iStep + 10;

	10: // Wait till read finish 

		IF NOT fbSoERead.Busy THEN
			fbSoERead.Execute			:= FALSE;
			IF fbSoERead.Error THEN
				wInitErrorCount 		:= wInitErrorCount + 1;
				// Count > 10 then go to error and wait for reset, if not wait in warning step
				IF wInitErrorCount > 10 THEN
					uiAdsErrId			:= fbSoERead.AdsErrId;
					uiSercosErrId		:= fbSoERead.SercosErrId;
					iStep				:= 1000;								// Error step
				ELSE
					iStep				:= 900;									// Warning step
				END_IF
			ELSE
				iStep 					:= iStep + 5;
			END_IF
		END_IF

	15: // Read Drive firmware version

		MEMCPY(ADR(S_0_0030_Value), (ADR(arr_S_0_0030_Value)+4), 62);
		iFWPos							:= FIND(S_0_0030_Value,': v') + 3;
		sDriveFW						:= DELETE(S_0_0030_Value, iFWPos -1,1);
		iFWLen							:= FIND(sDriveFW,'.');
		iFW_High						:= STRING_TO_INT(LEFT(sDriveFW, iFWLen-1));
		sDriveFW						:= DELETE(sDriveFW,iFWLen,1);
		iFWLen							:= FIND(sDriveFW,' ');
		iFW_Low							:= STRING_TO_INT(LEFT(sDriveFW, iFWLen-1));
		
		bDriveFirmware_GE_2_10 			:= iFW_High >= 2 AND iFW_Low >= 10;				// Check if firmware >= 2.10
		iStep	 						:= iStep + 5;		

	20: // Read P_0_0092 - Configured channel peak current

		fbSoERead.Idn 					:= P_0_IDN + 92;
		fbSoERead.Element				:= EC_SOE_ELEMENT_VALUE;
		fbSoERead.pDstBuf				:= ADR(P_0_0092_Value);
		fbSoERead.BufLen				:= SIZEOF(P_0_0092_Value);
		fbSoERead.Execute				:= TRUE;
		iStep 							:= iStep + 10;

	30: // Wait till read finish 

		IF NOT fbSoERead.Busy THEN
			fbSoERead.Execute			:= FALSE;
			IF fbSoERead.Error THEN
				wInitErrorCount 		:= wInitErrorCount + 1;
				// Count > 10 then go to error and wait for reset, if not wait in warning step
				IF wInitErrorCount > 10 THEN
					uiAdsErrId			:= fbSoERead.AdsErrId;
					uiSercosErrId		:= fbSoERead.SercosErrId;
					iStep				:= 1000;								// Error step
				ELSE
					iStep				:= 900;									// Warning step
				END_IF
			ELSE
				iStep 					:= iStep + 10;
			END_IF
		END_IF

	40: // Read P_0_0070 - Motor continuous stall torque

		fbSoERead.Idn 					:= P_0_IDN + 70;
		fbSoERead.Element				:= EC_SOE_ELEMENT_VALUE; 
		fbSoERead.pDstBuf				:= ADR(P_0_0070_Value);
		fbSoERead.BufLen 				:= SEL(bDriveFirmware_GE_2_10, 2, 4);		// In FW GE 2.10 size is 4
		fbSoERead.Execute				:= TRUE;
		iStep 							:= iStep + 10;

	50: // Wait till read finish 

		IF NOT fbSoERead.Busy THEN
			fbSoERead.Execute			:= FALSE;
			IF fbSoERead.Error OR P_0_0070_Value = 0 THEN						// P_0_0070_Value = 0 - probably linear motor or wrong motor data
				wInitErrorCount 		:= wInitErrorCount + 1;
				// Count > 10 then go to error and wait for reset, if not wait in warning step
				IF wInitErrorCount > 10 THEN
					uiAdsErrId			:= fbSoERead.AdsErrId;
					uiSercosErrId		:= fbSoERead.SercosErrId;
					iStep				:= 1000;								// Error step
				ELSE
					iStep				:= 900;									// Warning step
				END_IF
			ELSE
				iStep 					:= iStep + 10;
			END_IF
		END_IF

	60: // Read S_0_0111 - Motor continuous stall current

		fbSoERead.Idn 					:= S_0_IDN + 111;
		fbSoERead.Element				:= EC_SOE_ELEMENT_VALUE;
		fbSoERead.pDstBuf				:= ADR(S_0_0111_Value);
		fbSoERead.BufLen				:= SIZEOF(S_0_0111_Value);
		fbSoERead.Execute				:= TRUE;
		iStep 							:= iStep + 10;
		
	70: // Wait till read finish 

		IF NOT fbSoERead.Busy THEN
			fbSoERead.Execute			:= FALSE;
			IF fbSoERead.Error OR S_0_0111_Value = 0 THEN			// S_0_0111_Value = 0 - wrong motor data
				wInitErrorCount 		:= wInitErrorCount + 1;
				// Count > 10 then go to error and wait for reset, if not wait in warning step
				IF wInitErrorCount > 10 THEN
					uiAdsErrId			:= fbSoERead.AdsErrId;
					uiSercosErrId		:= fbSoERead.SercosErrId;
					iStep				:= 1000;								// Error step
				ELSE
					iStep				:= 900;									// Warning step
				END_IF
			ELSE
				iStep 					:= iStep + 10;
			END_IF
		END_IF

	80: // Read P_0_0093 - Configured channel current

		fbSoERead.Idn 					:= P_0_IDN + 93;
		fbSoERead.Element				:= EC_SOE_ELEMENT_VALUE;
		fbSoERead.pDstBuf				:= ADR(P_0_0093_Value);
		fbSoERead.BufLen				:= SIZEOF(P_0_0093_Value);
		fbSoERead.Execute				:= TRUE;
		iStep 							:= iStep + 10;
	
	90: // Wait till read finish 

		IF NOT fbSoERead.Busy THEN
			fbSoERead.Execute			:= FALSE;
			IF fbSoERead.Error THEN
				wInitErrorCount 		:= wInitErrorCount + 1;
				// Count > 10 then go to error and wait for reset, if not wait in warning step
				IF wInitErrorCount > 10 THEN
					uiAdsErrId			:= fbSoERead.AdsErrId;
					uiSercosErrId		:= fbSoERead.SercosErrId;
					iStep				:= 1000;								// Error step
				ELSE
					iStep				:= 900;									// Warning step
				END_IF
			ELSE
				iStep 					:= iStep + 10;							
			END_IF
		END_IF
		
	100: // Read data from unit finished - we can calculate params

		rPeakCurrent 					:= DWORD_TO_REAL(P_0_0092_Value) / 1000.0;		// In [A]
		rSfCurrent 						:= rPeakCurrent / 1000.0;						// iTorque -1000..1000 --> - rPeakCurrent .. rPeakCurrent
		rContinuousStallTorque 			:= DWORD_TO_REAL(P_0_0070_Value) / 100;
		rContinuousStallCurrent 		:= DWORD_TO_REAL(S_0_0111_Value) / 1000;
		IF rContinuousStallCurrent <> 0 THEN
			rSfTorque	 				:= rContinuousStallTorque / rContinuousStallCurrent;
		END_IF
		rWarningCurrent 				:= DWORD_TO_REAL(P_0_0093_Value) / 1000;
		iStep 							:= 200;

	200: // Read cycle time - we need it for I2T calculations

		fbGETCURTASKINDEX(index => BIndex);
		IF BIndex <> 0 THEN
			iStep						:= iStep + 10;
		END_IF

	210:

		rCycleTime 						:= UDINT_TO_REAL(_TaskInfo[BIndex].CycleTime) / 10000.0;	// Scale to [ms]
		rI2T_Window 					:= TIME_TO_REAL(tI2T_Window);
		wNoOfCycles						:= REAL_TO_WORD(rI2T_Window / rCycleTime);
		// Time window too short
		IF wNoOfCycles < 100 THEN
			iStep						:= 1000;								// Error step
		ELSE
			wProbeCyclesCount 			:= wNoOfCycles / 100;
			iStep						:= 300;
		END_IF

	300: // Calculations	

		ACT_I2T();
	
	900: // Warning - wait and repeat read - problem during read motor data, i.e. EtherCAT doesn't work yet

		IF tonWait.Q THEN
			iStep 						:= 0;	// Repeat initialization phase 
		END_IF
		
	1000: // Error - wait for reset 
		;

END_CASE
//===============================================================

bError		 							:= iStep = 1000;
bInitialized 							:= iStep >= 300 AND NOT bError;
ACT_Calculations();

//========================= Warning =============================
bWarning								:= rCurrentF > rWarningCurrent;

//===================== Limit output torque =====================
IF rTorqueLimit < rTorqueLimitLow THEN
	uiBipolarTorqueLimitValue 			:= REAL_TO_UINT(rTorqueLimitHigh);			// Secure against 0 value - probably empty var connected to input
ELSE
	uiBipolarTorqueLimitValue 			:= REAL_TO_UINT(LIMIT(rTorqueLimitLow,rTorqueLimit,rTorqueLimitHigh)) * 10;
END_IF

//====================== Call SoE read FB =======================
fbSoERead(	NetId:= '',
			Timeout:= T#1s,
			Axis:= Axis);

ACTION ACT_Calculations:
//============== Raw values - always avaliable ==================
rTorquePerc								:= LREAL_TO_REAL(Axis.NcToPlc.ActTorque); 		// [%]
rTorqueRAW 								:= rTorquePerc * 10;							// -1000 .. 1000 - RAW values the same as process image
//===================== Filter current value ====================
fbFilterEx(rIn:= rTorqueRAW, tTimeConstant:= T#1S);

// Calculations	- possible only with params
IF bInitialized THEN
	rCurrent 							:= rTorqueRAW * rSfCurrent;
	rTorque 							:= rCurrent * rSfTorque;
	rCurrentF 							:= fbFilterEx.rOut * rSfCurrent;
	rTorqueF 							:= rCurrentF * rSfTorque;
END_IF

//=============== Save torque and current max values ===============
IF ABS(rCurrentMax) < ABS(rCurrentF) THEN
	rTorquePercMax						:= rTorquePerc;
	rCurrentMax 						:= rCurrentF;
	rTorqueMax 							:= rTorqueF;
END_IF
END_ACTION

ACTION ACT_I2T:
//======================= One probe =============================
rCurrentPom 							:= rCurrentPom + ABS(rCurrent);
wCyclesCount							:= wCyclesCount + 1;
bCalculateI2T							:= FALSE;
IF wCyclesCount = wProbeCyclesCount THEN
	rCurrentAverage 					:= rCurrentPom / WORD_TO_REAL(wProbeCyclesCount);
	rCurrentPom							:= 0;
	wCyclesCount						:= 0;
	bCalculateI2T						:= TRUE;							
ELSIF wCyclesCount > wProbeCyclesCount THEN
	iStep 								:= 1000;
END_IF
//===============================================================

//==================== Recalculate I2T ==========================
IF bCalculateI2T THEN
	wNoOfProbes 						:= wNoOfProbes + 1;
	bBufferFull 						:= wNoOfProbes >= 100;
	MEMMOVE(ADR(arrI2TBuffer) + 4, ADR(arrI2TBuffer), SIZEOF(arrI2TBuffer) - 4);
	arrI2TBuffer[1]						:= rCurrentAverage;
	IF bBufferFull THEN
		rI2T_Nominal					:= 100.0 * rContinuousStallCurrent;
		rI2T_Actual						:= 0;
		FOR i := 1 TO 100 DO
			rI2T_Actual					:= rI2T_Actual + arrI2TBuffer[i];
		END_FOR
	ELSE
		rI2T_Nominal					:= wNoOfProbes * rContinuousStallCurrent;
		rI2T_Actual						:= rI2T_Actual + rCurrentAverage;
	END_IF
	rI2T								:= rI2T_Actual * 100 / rI2T_Nominal; // In [%]
//====================== Save I2T max value =====================
	IF rI2TMax < rI2T THEN
		rI2TMax							:= rI2T;
	END_IF
END_IF
//===============================================================
END_ACTION

ACTION ACT_Init_Reset:
//============== Reset max values and FB ========================
rtReset(CLK:= bReset);
// Reset I2T calculations when time window changed or reset CMD
IF rtReset.Q OR tI2T_Window <> tI2T_WindowOld THEN
	BIndex								:= 0;
	wProbeCyclesCount					:= 0;
	wCyclesCount						:= 0;
	wNoOfCycles							:= 0;
	wNoOfProbes							:= 0;
	i									:= 0;
	rCycleTime							:= 0;
	rI2T_Window							:= 0;
	rCurrentPom							:= 0;
	rCurrentAverage						:= 0;
	rI2T_Nominal						:= 0;
	rI2T_Actual							:= 0;
	rI2T								:= 0;
	rI2TMax								:= 0;
	MEMSET(ADR(arrI2TBuffer), 0, SIZEOF(arrI2TBuffer));
	bBufferFull							:= FALSE;
	bCalculateI2T						:= FALSE;
	// If there is no Error then recalculate time-dipendent variables
	IF NOT bError THEN
		iStep							:= 200;
	END_IF
	tI2T_WindowOld 						:= tI2T_Window;
END_IF

IF rtReset.Q OR bFirstCycle THEN
	fbSoERead.Execute					:= FALSE;
	bWarning	 						:= FALSE;
	bDriveFirmware_GE_2_10 				:= FALSE;
	uiAdsErrId		 					:= 0;
	uiSercosErrId	 					:= 0;
	rWarningCurrent 					:= 0;
	rTorquePerc 						:= 0;
	rTorquePercMax 						:= 0;
	rTorque 							:= 0;
	rTorqueF 							:= 0;
	rTorqueMax 							:= 0;
	rCurrent 							:= 0;
	rCurrentF 							:= 0;
	rCurrentMax 						:= 0;
	rTorqueRAW 							:= 0;
	rContinuousStallTorque 				:= 0;
	rContinuousStallCurrent 			:= 0;
	rPeakCurrent 						:= 0;
	rSfTorque 							:= 0;
	rSfCurrent							:= 0;
	iStep								:= 0;
	wInitErrorCount						:= 0;
	MEMSET(ADR(arr_S_0_0030_Value), 0, SIZEOF(arr_S_0_0030_Value));
	S_0_0030_Value						:= '';
	P_0_0092_Value						:= 0;
	P_0_0093_Value						:= 0;
	P_0_0070_Value						:= 0;
	S_0_0111_Value						:= 0;
	bFirstCycle	 						:= FALSE;
END_IF
END_ACTION

END_FUNCTION_BLOCK

// ---- POUs/FB/POUsAxisOnline/AX8000/F_AX8xErrMsg_1.TcPOU
//==================================================================================================
//							Beckhoff Automation Poland
//								7.12.2018
//		Funkcja konwertujaca nr bledu na opis
// 	v1.0	|| TC v 3.1.4022.27	|| - pierwsza wersja
//==================================================================================================
FUNCTION F_AX8xErrMsg_1 : STRING(255)
VAR_INPUT
	uiDriveError : UINT;
END_VAR

IF uiDriveError < 1 THEN
	F_AX8xErrMsg := '';
	RETURN;
END_IF

CASE uiDriveError OF
	16#2220: F_AX8xErrMsg:= '2220 =  Continuous over current (device internal)';
	16#2310: F_AX8xErrMsg:= '2310 =  Continuous over current (device output side)';
	16#2330: F_AX8xErrMsg:= '2330 = Earth leakage (motor-side)';
	16#2340: F_AX8xErrMsg:= '2340 =  Short circuit (motor-side)';
	16#2380: F_AX8xErrMsg:= '2380 =  Continuous over current (device output side) Phase U';
	16#2381: F_AX8xErrMsg:= '2381 =  Continuous over current (device output side) Phase V';
	16#2382: F_AX8xErrMsg:= '2382 =  Continuous over current (device output side) Phase W';
	16#2383: F_AX8xErrMsg:= '2383 =  Phase U current offset out of range';
	16#2384: F_AX8xErrMsg:= '2384 =  Phase V current offset out of range';
	16#2385: F_AX8xErrMsg:= '2385 =  Phase W current offset out of range';
	16#3110: F_AX8xErrMsg:= '3110 =  Mains over-voltage';
	16#3120: F_AX8xErrMsg:= '3120 =  Mains under-voltage';
	16#3130: F_AX8xErrMsg:= '3130 =  Phase failure';
	16#3180: F_AX8xErrMsg:= '3180 =  Phase failure motor or Mains voltage over brake resistor operating voltage';
	16#3181: F_AX8xErrMsg:= '3181 =  Phase frequency (motor-side) raised above 600 Hz or Wrong mains type';
	16#3182: F_AX8xErrMsg:= '3182 =  Velocity actual Value raised above the max channel accepted velocity';
	16#3183: F_AX8xErrMsg:= '3183 = The bipolar velocity limit is higher than 1/4 of position range limit per EtherCAT Sync1 cycle.';
	16#3210: F_AX8xErrMsg:= '3210 =  DC link over-voltage';
	16#3220: F_AX8xErrMsg:= '3220 =  DC link undervoltage';
	16#3280: F_AX8xErrMsg:= '3280 =  DC link is not ready or  Device DC link over-voltage';
	16#4110: F_AX8xErrMsg:= '4110 =  Excess ambient temperature';
	16#4210: F_AX8xErrMsg:= '4210 =  Excess temperature device';
	16#4310: F_AX8xErrMsg:= '4310 =  Drive overtemperature shut down';
	16#4380: F_AX8xErrMsg:= '4380 =  Fan speed seems to be zero.';
	16#5112: F_AX8xErrMsg:= '5112 =  Supply low voltage: supply +24V';
	16#5180: F_AX8xErrMsg:= '5180 =  Output stage STO active.';
	16#5181: F_AX8xErrMsg:= '5181 =  Power supply status,  torque off order';
	16#5182: F_AX8xErrMsg:= '5182 =  Power supply status inactive';
	16#5183: F_AX8xErrMsg:= '5183 =  Power supply status,  NC handling order';
	16#5184: F_AX8xErrMsg:= '5184 =  Supply DC-link circuit is not ready';
	16#5185: F_AX8xErrMsg:= '5185 =  Power supply status,  non-regenerative brake order';
	16#5186: F_AX8xErrMsg:= '5186 =  Power supply status,  regenerative brake order';
	16#5187: F_AX8xErrMsg:= '5187 =  Power supply communication is not established';
	16#5190: F_AX8xErrMsg:= '5190 =  Test 5V supply failed';
	16#5192: F_AX8xErrMsg:= '5192 =  Supply high voltage: supply +24V';
	16#5441: F_AX8xErrMsg:= '5441 =  Positive limit switch active';
	16#5442: F_AX8xErrMsg:= '5442 =  Negative limit switch active';
	16#5580: F_AX8xErrMsg:= '5580 =  Read failure EEPROM';
	16#5581: F_AX8xErrMsg:= '5581 =  Checksum failure EEPROM';
	16#5582: F_AX8xErrMsg:= '5582 =  EEPROM contains blank Data';
	16#5583: F_AX8xErrMsg:= '5583 =  Unexpected EEPROM';
	16#5584: F_AX8xErrMsg:= '5584 =  EEPROM contains blank Data';
	16#5585: F_AX8xErrMsg:= '5585 =  Unexpected EEPROM';
	16#5586: F_AX8xErrMsg:= '5586 =  Restored Errormessages from persistant memory';
	16#5587: F_AX8xErrMsg:= '5587 =  Missing factory settings in eeprom';
	16#5588: F_AX8xErrMsg:= '5588 =  Missing ids in eeprom display board';
	16#5589: F_AX8xErrMsg:= '5589 =  Read failure eeprom display board';
	16#5590: F_AX8xErrMsg:= '5590 =  Detected incompatible Pcb';
	16#5591: F_AX8xErrMsg:= '5591 =  Identity incompatible to a Pcb';
	16#5592: F_AX8xErrMsg:= '5592 =  FirmwareIndex is incompatible to this Firmware.';
	16#5593: F_AX8xErrMsg:= '5593 =  Structure Version is incompatible to this Firmware';
	16#5594: F_AX8xErrMsg:= '5594 =  Simulating persistent data features.';
	16#5595: F_AX8xErrMsg:= '5595 =  Modulo remainder will not be stored.';
	16#5596: F_AX8xErrMsg:= '5596 =  Storing of persistant data failed.';
	16#6010: F_AX8xErrMsg:= '6010 =  Software reset (watchdog)';
	16#6080: F_AX8xErrMsg:= '6080 =  Failure config bits';
	16#6180: F_AX8xErrMsg:= '6180 =  Internal Software Error Type A';
	16#6181: F_AX8xErrMsg:= '6181 =  Internal Software Error Type B';
	16#6182: F_AX8xErrMsg:= '6182 =  Internal Software Error Type C';
	16#6183: F_AX8xErrMsg:= '6183 =  Internal Watchdog Error';
	16#6190: F_AX8xErrMsg:= '6190 =  Init Timeout';
	16#6310: F_AX8xErrMsg:= '6310 =  Loss of parameters';
	16#6320: F_AX8xErrMsg:= '6320 =  Parameter error';
	16#6380: F_AX8xErrMsg:= '6380 =  Parameter Interpolator: Illegal Interpolation sub mode select or  Parameters x with parametrized y is too low.';
	16#6381: F_AX8xErrMsg:= '6381 =  Parameter x with parametrized y is too high';
	16#6382: F_AX8xErrMsg:= '6382 =  Illegal Slotconfiguration. Slot is empty.';
	16#6383: F_AX8xErrMsg:= '6383 =  Illegal Slotconfiguration. Double Feedback Selection.';
	16#6384: F_AX8xErrMsg:= '6384 =  Illegal Slotconfiguration. Slot has to be empty.';
	16#6385: F_AX8xErrMsg:= '6385 =  Parameter Interpolator. Operation Mode does not match';
	16#6386: F_AX8xErrMsg:= '6386 =  Parameter Interpolator: Illegal NC-Task cycle time';
	16#6387: F_AX8xErrMsg:= '6387 =  Parameter Motor. The configured DCLink Max Voltage is higher than the Motor Max Voltage.';
	16#6388: F_AX8xErrMsg:= '6388 =  Parameter Torque Control: The value in Object 0x%x/%x is higher than the Motor peak current (0x%x/%x).';
	16#6389: F_AX8xErrMsg:= '6389 =  Parameter Torque Control: The value in Object 0x%x/%x is higher than the Configured peak current (0x%x/%x).';
	16#6390: F_AX8xErrMsg:= '6390 =  Factor Group Parameters: Feed constant illegal feed';
	16#6391: F_AX8xErrMsg:= '6391 =  Factor Group Parameters: Feed constant illegal shaft revolutions';
	16#6392: F_AX8xErrMsg:= '6392 =  Factor Group Parameters: Gear ratio illegal Motor shaft revolutions';
	16#6393: F_AX8xErrMsg:= '6393 =  Factor Group Parameters: Gear ratio illegal Driving shaft revolutions';
	16#6394: F_AX8xErrMsg:= '6394 =  Factor Group Parameters: Position encoder resolution illegal encoder increments';
	16#6395: F_AX8xErrMsg:= '6395 =  Factor Group Parameters: Position encoder resolution illegal motor revolutions';
	16#6396: F_AX8xErrMsg:= '6396 =  additional Factor Group Parameters: Feed constant illegal feed';
	16#6397: F_AX8xErrMsg:= '6397 =  additional Factor Group Parameters: Feed constant illegal shaft revolutions';
	16#6398: F_AX8xErrMsg:= '6398 =  additional Factor Group Parameters: Gear ratio illegal Motor shaft revolutions';
	16#6399: F_AX8xErrMsg:= '6399 =  additional Factor Group Parameters: Gear ratio illegal Driving shaft revolutions';
	16#7111: F_AX8xErrMsg:= '7111 =  Failure brake chopper';
	16#7112: F_AX8xErrMsg:= '7112 =  Over current brake chopper';
	16#7122: F_AX8xErrMsg:= '7122 =  Motor error or commutation malfunction';
	16#7180: F_AX8xErrMsg:= '7180 =  Motor brake: Current monitoring error. Or  Brake resistor not found';
	16#7181: F_AX8xErrMsg:= '7181 =  Motor thermal utilization has reached the warning level.  Or  Brake resistor power overload by DC link over-voltage';
	16#7182: F_AX8xErrMsg:= '7182 =  Motor thermal utilization has left the warning level. Or  Wrong xml file';
	16#7183: F_AX8xErrMsg:= '7183 =  Motor thermal utilization has reached the Error Level';
	16#7184: F_AX8xErrMsg:= '7184 =  Motor overload shut down';
	16#7185: F_AX8xErrMsg:= '7185 =  Motor overtemperature shut down';
	16#7186: F_AX8xErrMsg:= '7186 = Detected moving axis on enable transition.';
	16#7320: F_AX8xErrMsg:= '7320 =  HpfDsl: Encoder error (position invalid)';
	16#7380: F_AX8xErrMsg:= '7380 =  Current sensor motor phase U or HpfDsl: Encoder start sequence failed';
	16#7381: F_AX8xErrMsg:= '7381 =  Current sensor motor phase V or HpfDsl: Encoder shutdown failed';
	16#7382: F_AX8xErrMsg:= '7382 =  Current sensor motor phase W or HpfDsl: Parameter access error';
	16#7383: F_AX8xErrMsg:= '7383 =  HpfDsl: Internal error';
	16#7384: F_AX8xErrMsg:= '7384 =  HpfDsl: Cyclic monitoring error';
	16#7385: F_AX8xErrMsg:= '7385 =  HpfDsl: Encoder file processing';
	16#7386: F_AX8xErrMsg:= '7386 =  HpfDsl: Found no encoder (No link to an encoder)!';
	16#7580: F_AX8xErrMsg:= '7580 =  I2C_communication_failure';
	16#8180: F_AX8xErrMsg:= '8180 =  System restart or sync lost';
	16#8181: F_AX8xErrMsg:= '8181 =  Lost Distributed clocks Sync';
	16#8182: F_AX8xErrMsg:= '8182 =  EtherCAT Statemachine shutdown with enabled Axis';
	16#8183: F_AX8xErrMsg:= '8183 =  Controlword output cycle counter monitoring';
	16#8480: F_AX8xErrMsg:= '8480 = Overspeed error';
	16#8611: F_AX8xErrMsg:= '8611 = Following error';
	16#8680: F_AX8xErrMsg:= '8680 =  Position Demand Value outside of the specified Position Range Limits';
	16#8780: F_AX8xErrMsg:= '8780 =  Configured Sync1 Cycle Time is above Maximum';
	16#8781: F_AX8xErrMsg:= '8781 =  Configured Sync1 Cycle Time is below Minimum';
	16#8782: F_AX8xErrMsg:= '8782 =  Configured Sync1 Cycle Time is not a multiple of the Sync0 Cycle Time';
	16#8783: F_AX8xErrMsg:= '8783 =  Configured Sync0 Cycle Time is not legal';
	16#638A: F_AX8xErrMsg:= '638A =  The Axis seems not to be parameterised.';
	16#638B: F_AX8xErrMsg:= '638B =  Parameter Torque Current curve: Unable to calculate Torque Current curve.';
	16#638C: F_AX8xErrMsg:= '638C =  Motor type does not match';
	16#638D: F_AX8xErrMsg:= '638D =  Connected Motor is compatible to the configured Motor';
	16#638E: F_AX8xErrMsg:= '638E =  The Motor brake is automatically unlocked';
	16#638F: F_AX8xErrMsg:= '638F =  Parameter Torque Control: The value in Object 0x%x/%x is higher then the Motor maximum voltage slope (0x%x/%x).';
	16#639A: F_AX8xErrMsg:= '639A =  additional Factor Group Parameters: Position encoder resolution illegal encoder increments';
	16#639B: F_AX8xErrMsg:= '639B =  additional Factor Group Parameters: Position encoder resolution illegal motor revolutions';
	16#639C: F_AX8xErrMsg:= '639C =  Velocity factor illegal. A possible Value would be %u/%u.';
	16#639D: F_AX8xErrMsg:= '639D =  Acceleration factor illegal. A possible Value would be %u/%u.';
	16#639E: F_AX8xErrMsg:= '639E =  Scaling index object 0x%x does not fit the Factor group parameters for the first Encoder';
	16#639F: F_AX8xErrMsg:= '639F =  Scaling index object 0x%x does not fit the Factor group parameters for the second Encoder';
	16#63A0: F_AX8xErrMsg:= '63A0 =  Motor or Primary Feedback changed';
	16#63A1: F_AX8xErrMsg:= '63A1 =  Secondary Feedback changed';
	16#63A2: F_AX8xErrMsg:= '63A2 =  Offset position actual value: No position offset existing in source "encoder memory"';
	16#63A3: F_AX8xErrMsg:= '63A3 =  Offset additional position actual value: No position offset existing in source "encoder memory"';
	16#63A4: F_AX8xErrMsg:= '63A4 =  Offset position actual value: No position offset existing in source "drive memory"';
	16#63A5: F_AX8xErrMsg:= '63A5 =  Offset additional position actual value: No position offset existing in source "drive memory"';
	16#63A6: F_AX8xErrMsg:= '63A6 =  Jerk factor illegal. A possible Value would be %u/%u.';
	16#63A7: F_AX8xErrMsg:= '63A7 =  The range %u of the Position range limit is below the minimum accepted value of %u.';
	16#63A8: F_AX8xErrMsg:= '63A8 =  Position range limit Inc with remainder is not supported for primary feedback.';
	16#63A9: F_AX8xErrMsg:= '63A9 =  Position range limit Inc with remainder is not supported for secondary feedback.';
	16#63AA: F_AX8xErrMsg:= '63AA =  Object 0x%X/%X changed in EtherCAT SafeOP or OP.';
	16#8A80: F_AX8xErrMsg:= '8A80 =  Illegal Modes of Operation';
	16#8A81: F_AX8xErrMsg:= '8A81 =  Illegal Modes of Operation change';
	16#A000: F_AX8xErrMsg:= 'A000 =  Transition Pre-Op to Safe-Op not successful. Sync Manager Length Error.';
	16#A001: F_AX8xErrMsg:= 'A001 =  Transition Pre-Op to Safe-Op not successful. Sync Manager Address Error.';
	16#A002: F_AX8xErrMsg:= 'A002 =  Transition Pre-Op to Safe-Op not successful. Sync Manager Settings Error.';
	16#A003: F_AX8xErrMsg:= 'A003 =  Transition Pre-Op to Safe-Op not successful. Sync Manager Address Range overlap.';
	16#A004: F_AX8xErrMsg:= 'A004 =  Sync Manager is disabledand has a Size unequal zero.';
	16#A010: F_AX8xErrMsg:= 'A010 =  SDO Complete Access Error: Object 0x%x/%x';
	16#A011: F_AX8xErrMsg:= 'A011 =  RxPdo Mapping Error: Unable to map Object (not possible).';
	16#A012: F_AX8xErrMsg:= 'A012 =  TxPdo Mapping Error: Unable to map Object (not possible).';
	16#A013: F_AX8xErrMsg:= 'A013 =  RxPdo Mapping Error: Double Mapping of Object.';
	16#A014: F_AX8xErrMsg:= 'A014 =  TxPdo Mapping Error: Double Mapping of Object.';
	16#A015: F_AX8xErrMsg:= 'A015 =  RxPdo Mapping Error: Unable to map Object (no Mappings left).';
	16#A016: F_AX8xErrMsg:= 'A016 =  TxPdo Mapping Error: Unable to map Object (no Mappings left).';
	16#A017: F_AX8xErrMsg:= 'A017 =  RxPdo Mapping Error: Object always has to be mapped.';
	16#A018: F_AX8xErrMsg:= 'A018 =  TxPdo Mapping Error: Object 0x%x/%x always has to be mapped.';
	16#A019: F_AX8xErrMsg:= 'A019 =  RxPdo Mapping Error: Object has to be mapped because of modes of operation.';
	16#A01A: F_AX8xErrMsg:= 'A01A =  TxPdo Mapping Error: Object has to be mapped because of modes of operation.';
	16#A01B: F_AX8xErrMsg:= 'A01B =  RxPdo BitMapping Error: Object 0x%x/%x is not next to Object 0x%x/%x. (SyncManager %u)';
	16#A01C: F_AX8xErrMsg:= 'A01C =  TxPdo BitMapping Error: Object 0x%x/%x is not next to Object 0x%x/%x. (SyncManager %u)';
	16#A01D: F_AX8xErrMsg:= 'A01D =  RxPdo BitMapping Error: Can not Transform Bit-Mappings to Byte-Mappings. (SyncManager %u)';
	16#A01E: F_AX8xErrMsg:= 'A01E =  TxPdo BitMapping Error: Can not Transform Bit-Mappings to Byte-Mappings. (SyncManager %u)';
	16#A080: F_AX8xErrMsg:= 'A080 =  Safe-Op is not possible because the local TwinCAT Runtime is in ConfigMode.';
	16#A081: F_AX8xErrMsg:= 'A081 =  Transition Pre-Op to Safe-Op not successful. Safetycard not detected.';
	16#A082: F_AX8xErrMsg:= 'A082 =  EtherCAT Slave Stack Error:';
	16#FF01: F_AX8xErrMsg:= 'FF01 =  Init Timeout or Error reaction forced: Generative brake order';
	16#FF02: F_AX8xErrMsg:= 'FF02 =  Error reaction forced: Non-generative brake order';
	16#FF03: F_AX8xErrMsg:= 'FF03 =  Error reaction forced: Brake chopper off';
	16#FF07: F_AX8xErrMsg:= 'FF07 =  Error reaction forced: Torque Off';
	16#FF08: F_AX8xErrMsg:= 'FF08 =  Error reaction forced: Shorted Coils Brake';
	16#FF09: F_AX8xErrMsg:= 'FF09 =  Error reaction forced: Open Loop Ramp';
	16#FF0A: F_AX8xErrMsg:= 'FF0A =  Error reaction forced: Closed Loop Ramp';
	16#FF0B: F_AX8xErrMsg:= 'FF0B =  Error reaction forced: NC handling';
	16#FF0C: F_AX8xErrMsg:= 'FF0C =  Error reaction TorqueOff with emergency brake';
	16#FFFC: F_AX8xErrMsg:= 'FFFC =  %s';
	16#FFFD: F_AX8xErrMsg:= 'FFFD =  Debug firmware.  Replace "As soon as possible"!';
	16#FFFE: F_AX8xErrMsg:= 'FFFE =  %s';
	16#FFFF: F_AX8xErrMsg:= 'FFFF =  Internal Error.   Additional Errorcode 0x%x';

ELSE
	F_AX8xErrMsg := UINT_TO_STRING(uiDriveError);
	F_AX8xErrMsg := concat(F_AX8xErrMsg, ' Unknown Error code');
END_CASE
F_AX8xErrMsg := F_AX8xErrMsg;

END_FUNCTION

// ---- POUs/FB/POUsAxisOnline/EL72xx/FB_HoldingBrakeCtrlEL72xx.TcPOU
//==================================================================================================
//							Beckhoff Automation Poland
//									11.07.2018
//	Blok funkcyjny kontroli luzownika w silniku podpietym do EL72xx. Mozliwy jest jedynie force unlock.
//	Dzialania na obiekcie:	: 8012:01 (MDP742) lub 2004:01 (DS402)
//
//  v1.0	|| TC v 3.1.4022.22		|| - pierwsza wersja
//==================================================================================================
FUNCTION_BLOCK FB_HoldingBrakeCtrlEL72xx
VAR_INPUT
	bForceUnlock					: BOOL;								// Rising/falling edhe executes CMD: Manual override (release) of the motor holding brake 
																		// and reset - if there is error - falling edge reinits FB
	stDriveRef						: ST_DriveRef;
END_VAR
VAR_OUTPUT
	bBusy							: BOOL;
	bError							: BOOL; 							// General error: parameter or CoE read.
	uiAdsErrId						: UINT;								// Forwarded output FB_CoERead_ByDriveRef
	uiCANopenErrId					: UINT;								// Forwarded output FB_CoERead_ByDriveRef
END_VAR
VAR
	//======================= Internal var ===========================
	iStep							: INT;								// Case instruction	
	wInitErrorCount					: WORD;								// Initialization error counter, if bigger then 10 then error
	wManualOverrideIndex			: WORD;								// Manual override (release) of the motor holding brake:
																		// MDP742: 8012:01
																		// DS402: 2004:01
	bDriveRefOK						: BOOL;								// stDriveRef contains necessary data to read CoE
	bExecute						: BOOL;
	bDS402Profile					: BOOL;								// Flag DS402
	bMDP742Profile					: BOOL;								// Flag MDP742	
	bInitialized					: BOOL;
	sDeviceName						: STRING;							// 
	sNo								: STRING(1);						// xxxxxxx-000Y - char Y	
	//=========================== FBs ================================																
	rtForceUnlock					: R_TRIG;
	ftForceUnlock					: F_TRIG;
	tonWait							: TON;								// Wait timer
	fbCoERead						: FB_CoERead_ByDriveRef;			// FB for read CoE parameters
	fbForceUnlock					: FB_CoEWrite_ByDriveRef;
END_VAR

//=================== Call triggers and timers ==================
tonWait(IN:= NOT tonWait.Q, PT:= T#1S);
rtForceUnlock(CLK:= bForceUnlock);
ftForceUnlock(CLK:= bForceUnlock);

//======= Check for parameter error - each cycle ================
bDriveRefOK 							:= (stDriveRef.nSlaveAddr <> 0) AND (stDriveRef.sNetId <> '');

//============= Read params and calculations ====================
CASE iStep OF
	
	0: // Read profile MDP 742 or DS 402:
	
			// We have to read device name Index 1008:0 - STRING
			// EL72x1-0000 --> MDP 742:
			// EL72x1-0001 --> DS 402:
	
		// Execute read only if DriveRef is OK
		IF bDriveRefOK THEN
			fbCoERead.nIndex			:= 16#1008;
			fbCoERead.nSubIndex			:= 0;
			fbCoERead.pDstBuf			:= ADR(sDeviceName);
			fbCoERead.cbBufLen			:= SIZEOF(sDeviceName);
			fbCoERead.bExecute			:= TRUE;
			iStep 						:= iStep + 10; 
		END_IF
	
	10:	// Wait till read finish
	
		IF NOT fbCoERead.bBusy THEN
			fbCoERead.bExecute			:= FALSE;
			IF fbCoERead.bError THEN
				wInitErrorCount 		:= wInitErrorCount + 1;
				// Count > 10 then go to error and wait for reset, if not wait in warning step
				IF wInitErrorCount > 10 THEN
					uiAdsErrId			:= fbCoERead.iAdsErrId;
					uiCANopenErrId		:= fbCoERead.iCANopenErrId;
					iStep				:= 1000;								// Error step
				ELSE
					iStep				:= 900;									// Warning step
				END_IF
			ELSE
				iStep 					:= iStep + 10;
			END_IF
		END_IF

	20: // Check last digit in device name 0 - MDP742, 1 - DS402
	
	sNo 								:=  MID(sDeviceName, 1, FIND(sDeviceName, '-') + 4);
	bMDP742Profile 						:= 	sNo = '0';
	bDS402Profile 						:= 	sNo = '1';
	// If 0 or 1 then go to next step, if other No - not implemented yet
	IF bMDP742Profile OR bDS402Profile THEN
		wManualOverrideIndex			:= SEL(bMDP742Profile, 16#2004, 16#8012);
		iStep 							:= 100;
	ELSE
		iStep							:= 1000;					// Error step
	END_IF
	
	100: // Initialized - holding brake control possible
		fbForceUnlock.bExecute			:= rtForceUnlock.Q OR ftForceUnlock.Q;
		IF fbForceUnlock.bBusy THEN
			iStep 						:= iStep + 10;
		END_IF

	110: // Wait till write finish
	
		IF NOT fbForceUnlock.bBusy THEN
			fbForceUnlock.bExecute		:= FALSE;
			IF fbForceUnlock.bError THEN
				uiAdsErrId				:= fbForceUnlock.iAdsErrId;
				uiCANopenErrId			:= fbForceUnlock.iCANopenErrId;
			ELSE
				iStep 					:= iStep - 10;
			END_IF
		END_IF
	
	900: // Warning - wait and repeat read - problem during read motor data, i.e. EtherCAT doesn't work yet
		IF tonWait.Q THEN
			iStep 						:= 0;	// Repeat initialization phase 
		END_IF
			  
	1000: // Error - wait for reset 
		IF ftForceUnlock.Q THEN
			uiAdsErrId					:= 0;
			uiCANopenErrId				:= 0;
			wInitErrorCount				:= 0;
			wManualOverrideIndex		:= 0;
			sDeviceName					:= '';
			sNo							:= '';
			bDS402Profile				:= FALSE;
			bMDP742Profile				:= FALSE;
			iStep						:= 0;
		END_IF
END_CASE
//===============================================================

bError		 							:= iStep = 1000;
bInitialized 							:= iStep >= 100 AND iStep < 900;

//================== Call CoE read/write FB =====================
fbCoERead(stDriveRef:= stDriveRef);

fbForceUnlock	(	stDriveRef				:= stDriveRef, 
					nIndex					:= wManualOverrideIndex, 
					nSubIndex				:= 16#01, 
					pSrcBuf					:= ADR(bForceUnlock), 
					cbBufLen				:= SIZEOF(bForceUnlock));
//===============================================================

END_FUNCTION_BLOCK

// ---- POUs/FB/POUsAxisOnline/EL72xx/FB_McAxisOnlineEL72xx.TcPOU
//==================================================================================================
//							Beckhoff Automation Poland
//									7.12.2018
//	Wszystkomajacy blok funkcyjny do sterowania osia, 
//	wymagane biblioteki: Tc2_EtherCAT, Tc2_MC2_Drive, Tc2_MC2
//  v1.1	|| TC v 3.1.4022.27		|| - dodane opisy bledow w formie zmiennych typu string
// 	v1.0 	|| TC v 3.1.4022.22	 	|| - first edition
//==================================================================================================
{attribute 'reflection'}
FUNCTION_BLOCK FB_McAxisOnlineEL72xx
VAR_IN_OUT
	stMcAxisOnline						: ST_McAxisOnline;
	Axis								: AXIS_REF;
END_VAR
VAR
	mcPower								: MC_Power;
	mcStop								: MC_Stop;
	mcHalt								: MC_Halt;
	mcStopSS1							: MC_Stop;
	mcStopSS2							: MC_Stop;
	mcReset								: MC_Reset;
	mcHome								: MC_Home;
	mcSetPosition						: MC_SetPosition;
	fbSetPositionOffset					: FB_CoEEL72xxSetPositionOffset;// Not Yet avaliable
	mcJog								: MC_Jog;

	mcMoveAbsolute						: MC_MoveAbsolute;
	mcMoveRelative						: MC_MoveRelative;
	mcMoveVelocity						: MC_MoveVelocity;
	mcMoveModulo						: MC_MoveModulo;
	mcMoveAbsolute2						: MC_MoveAbsolute;
	mcMoveRelative2						: MC_MoveRelative;
	mcMoveVelocity2						: MC_MoveVelocity;
	mcMoveModulo2						: MC_MoveModulo;

	fbMotorMonitoring					: FB_MotorMonitoringEL72xx;
	fbHoldingBrakeCtrl					: FB_HoldingBrakeCtrlEL72xx;
	fbNcLimitSwitch						: FB_NcSWLimitSwitchCtrl;
	tonGetDriveDiag						: TON;
	fbReadChannelErrorCode				: FB_ReadChannelErrorCodeEL72xx;
	
	mcReadDriveAddress					: MC_ReadDriveAddress;
	mcReadParameterSet					: MC_ReadParameterSet;
	fbGetDriveRef						: FB_GetDriveRef;

	// Internal
	bInitialized						: BOOL;
	bCommError							: BOOL;
	bReadParameterError					: BOOL;
	bInitError							: BOOL;
	bDriveError							: BOOL;
	bFBError							: BOOL;
	
// Initialization
	iInitStep							: INT;
	bInitializationError				: BOOL;
	wInitializationErrorCounter			: WORD;
	bDriveAddressReady					: BOOL;
	bDriveRefReady						: BOOL;
	bReadParameterSetReady				: BOOL;
	tonDelay							: TON;
// Re init
	udiOnlineChangeCntOld				: UDINT;
	bOnlineChangeDetected				: BOOL;
	bReInit								: BOOL;
	bReInitialized						: BOOL;
	bReInitializationError				: BOOL;
	{attribute 'instance-path'}
	{attribute 'noinit'}
	sInstancePath						: STRING;
END_VAR

// Device dependent initialization 
ACT_Initialization();
// Device independent commands, mostly NC 
ACT_States();
ACT_SWLimitSwitch();
ACT_Stop();
ACT_Power();
ACT_Homing();
ACT_Jog();
ACT_Move();
ACT_Reset();
ACT_SetPosition();
// Device dependent commands
// Motor monitoring possible only with real axis
IF NOT Axis.Status.OpMode.SimulationAxis THEN
	ACT_MotorMonitoring();
END_IF
// Device dependent commands, possible only on real axis after complete initialization
IF bInitialized AND NOT Axis.Status.OpMode.SimulationAxis THEN
	ACT_SetPositionIO();
	ACT_DriveDiag();
	ACT_HoldingBrakeCtrl();
END_IF

// Device independent error collection
ACT_ErrorCollection();

ACTION ACT_DriveDiag:
// Auto update when drive error
tonGetDriveDiag(IN:= stMcAxisOnline.stError.bDriveError AND NOT tonGetDriveDiag.Q, PT:= T#5S, Q=> , ET=> );

fbReadChannelErrorCode(	bExecute				:= stMcAxisOnline.stChannelErrorCode.bExecute OR tonGetDriveDiag.Q,
						stDriveRef				:= stMcAxisOnline.stDriveRef,
						bBusy					=> stMcAxisOnline.stChannelErrorCode.bBusy,
						bError					=> stMcAxisOnline.stChannelErrorCode.bError,
						uiAdsErrId				=> stMcAxisOnline.stChannelErrorCode.uiAdsErrId,
						uiCANopenErrId			=> stMcAxisOnline.stChannelErrorCode.uiSecErrId,
						uiChannelErrorCode		=> stMcAxisOnline.stChannelErrorCode.uiChannelErrorCode,
						uiChannelErrorCodeHex	=> stMcAxisOnline.stChannelErrorCode.uiChannelErrorCodeHex);
END_ACTION

ACTION ACT_ErrorCollection:
// Error flags
stMcAxisOnline.stError.bDriveError					:= Axis.Status.DriveDeviceError;

stMcAxisOnline.stError.bNcError						:= Axis.Status.Error;

stMcAxisOnline.stError.bFBError						:= stMcAxisOnline.mcPower.bError OR stMcAxisOnline.mcReset.bError OR stMcAxisOnline.mcHome.bError OR stMcAxisOnline.mcJog.bError
													OR stMcAxisOnline.mcHalt.bError OR stMcAxisOnline.mcStop.bError OR stMcAxisOnline.mcSS1.bError OR stMcAxisOnline.mcSS2.bError
													OR stMcAxisOnline.mcMoveAbsolute.bError OR stMcAxisOnline.mcMoveRelative.bError OR stMcAxisOnline.mcMoveVelocity.bError OR stMcAxisOnline.mcMoveModulo.bError
													OR stMcAxisOnline.mcMoveAbsolute2.bError OR stMcAxisOnline.mcMoveRelative2.bError OR stMcAxisOnline.mcMoveVelocity2.bError OR stMcAxisOnline.mcMoveModulo2.bError
													OR stMcAxisOnline.stNcLimitSwitch.bError OR stMcAxisOnline.mcSetPosition.bError;
									
stMcAxisOnline.stError.bCommunicationError			:= stMcAxisOnline.stChannelErrorCode.bError OR stMcAxisOnline.stSetPositionOffset.bError OR stMcAxisOnline.stMotorMonitoring.bError OR stMcAxisOnline.stHoldingBrake.bError;

stMcAxisOnline.stError.bError						:= stMcAxisOnline.stError.bDriveError OR stMcAxisOnline.stError.bNcError OR stMcAxisOnline.stError.bFBError OR stMcAxisOnline.stError.bCommunicationError;
stMcAxisOnline.bError								:= stMcAxisOnline.stError.bError; // Forward one stage up

// Error codes
stMcAxisOnline.stError.uiDriveErrorID 				:= stMcAxisOnline.stChannelErrorCode.uiChannelErrorCode;
stMcAxisOnline.stError.uiDriveErrorIDHex 			:= stMcAxisOnline.stChannelErrorCode.uiChannelErrorCodeHex;

stMcAxisOnline.stError.udiNcErrorID 				:= Axis.Status.ErrorID;
stMcAxisOnline.stError.udiNcErrorIDHex 				:= Axis.Status.ErrorID;
	

stMcAxisOnline.stError.udiFBErrorID 				:= 	stMcAxisOnline.mcPower.udiErrorID + 
														stMcAxisOnline.mcReset.udiErrorID + 
														stMcAxisOnline.mcHome.udiErrorID + 
														stMcAxisOnline.mcJog.udiErrorID +
														stMcAxisOnline.mcHalt.udiErrorID + 
														stMcAxisOnline.mcStop.udiErrorID + 
														stMcAxisOnline.mcSS1.udiErrorID + 
														stMcAxisOnline.mcSS2.udiErrorID +
														stMcAxisOnline.mcMoveAbsolute.udiErrorID + 
														stMcAxisOnline.mcMoveRelative.udiErrorID + 
														stMcAxisOnline.mcMoveVelocity.udiErrorID + 
														stMcAxisOnline.mcMoveModulo.udiErrorID +
														stMcAxisOnline.mcMoveAbsolute2.udiErrorID + 
														stMcAxisOnline.mcMoveRelative2.udiErrorID + 
														stMcAxisOnline.mcMoveVelocity2.udiErrorID + 
														stMcAxisOnline.mcMoveModulo2.udiErrorID +
														stMcAxisOnline.stNcLimitSwitch.udiErrorID + 
														stMcAxisOnline.mcSetPosition.udiErrorID;

stMcAxisOnline.stError.udiFBErrorIDHex 				:= stMcAxisOnline.stError.udiFBErrorID;

stMcAxisOnline.stError.udiErrorID					:= stMcAxisOnline.stSetPositionOffset.udiErrorID;
stMcAxisOnline.stError.uiAdsErrorID					:= stMcAxisOnline.stChannelErrorCode.uiAdsErrId + stMcAxisOnline.stMotorMonitoring.uiAdsErrId + stMcAxisOnline.stHoldingBrake.uiAdsErrId;
stMcAxisOnline.stError.uiSecErrorID					:= stMcAxisOnline.stChannelErrorCode.uiSecErrId + stMcAxisOnline.stMotorMonitoring.uiSecErrId + stMcAxisOnline.stHoldingBrake.uiSecErrId;

stMcAxisOnline.stError.sNcError						:= F_AxErrMsg(stMcAxisOnline.stError.udiNcErrorID);
stMcAxisOnline.stError.sDriveError					:= F_EL72ErrMsg(stMcAxisOnline.stError.uiDriveErrorID);
END_ACTION

ACTION ACT_HoldingBrakeCtrl:
fbHoldingBrakeCtrl(bForceUnlock		:= stMcAxisOnline.stHoldingBrake.bForceUnlock,
					stDriveRef			:= stMcAxisOnline.stDriveRef,
					bBusy				=> stMcAxisOnline.stHoldingBrake.bBusy,
					bError				=> stMcAxisOnline.stHoldingBrake.bError,
					uiAdsErrId			=> stMcAxisOnline.stHoldingBrake.uiAdsErrId,
					uiCANopenErrId		=> stMcAxisOnline.stHoldingBrake.uiSecErrId);
END_ACTION

ACTION ACT_Homing:
mcHome(		Axis						:= Axis,
			Execute						:= stMcAxisOnline.mcHome.bExecute,
			Position					:= stMcAxisOnline.mcHome.lrPosition,
			HomingMode					:= stMcAxisOnline.mcHome.eHomingMode,
			BufferMode					:= stMcAxisOnline.mcHome.eBufferMode,
			Options						:= stMcAxisOnline.mcHome.stOptions,
			bCalibrationCam				:= stMcAxisOnline.mcHome.bCalibrationCam,
			Done						=> stMcAxisOnline.mcHome.bDone,
			Busy						=> stMcAxisOnline.mcHome.bBusy,
			Active						=> stMcAxisOnline.mcHome.bActive,
			CommandAborted				=> stMcAxisOnline.mcHome.bCommandAborted,
			Error						=> stMcAxisOnline.mcHome.bError,
			ErrorID						=> stMcAxisOnline.mcHome.udiErrorID);
END_ACTION

ACTION ACT_Initialization:
// bInitialized flag is set just once. 
// bReInitialized ise set each time we do online change or request reinit operation
// bDriveAddressReady, bReadParameterSetReady, bDriveRefReady - set just once after successed read

// Online change detection
bOnlineChangeDetected					:= udiOnlineChangeCntOld <> _AppInfo.OnlineChangeCnt;
udiOnlineChangeCntOld 					:= _AppInfo.OnlineChangeCnt;
// Reset init
IF bReInit OR bOnlineChangeDetected THEN
	iInitStep							:= 0;
END_IF

//Initialization process
CASE iInitStep OF
	0:	// Read Drive Address
		
		stMcAxisOnline.mcReadDriveAddress.bExecute	:=	 TRUE;
		iInitStep						:= iInitStep + 10;
		
	10: // Wait for data
	
		IF NOT stMcAxisOnline.mcReadDriveAddress.bBusy THEN
			stMcAxisOnline.mcReadDriveAddress.bExecute	:=	 FALSE;
			IF stMcAxisOnline.mcReadDriveAddress.bDone THEN
				iInitStep 				:= iInitStep + 10;
				bDriveAddressReady 		:= TRUE;
			ELSE
				iInitStep 				:= 1000;		// Error step
			END_IF
		END_IF
		
	20:	// Read Parameter Set
		
		stMcAxisOnline.mcReadParameterSet.bExecute		:=	 TRUE;
		iInitStep						:= iInitStep + 10;
		
	30: // Wait for data
	
		IF NOT stMcAxisOnline.mcReadParameterSet.bBusy THEN
			stMcAxisOnline.mcReadParameterSet.bExecute	:=	 FALSE;
			IF stMcAxisOnline.mcReadParameterSet.bDone THEN
				iInitStep 				:= iInitStep + 10;
				bReadParameterSetReady 	:= TRUE;
			ELSE
				iInitStep 				:= 1000;		// Error step
			END_IF
		END_IF	
	
	40:	// Get Drive Ref
		
		stMcAxisOnline.stGetDriveRef.bExecute		:=	 TRUE;
		iInitStep						:= iInitStep + 10;
		
	50: // Wait for data
	
		IF NOT stMcAxisOnline.stGetDriveRef.bBusy THEN
			stMcAxisOnline.stGetDriveRef.bExecute	:=	 FALSE;
			IF NOT stMcAxisOnline.stGetDriveRef.bError THEN
				iInitStep 				:= iInitStep + 10;
				bDriveRefReady 			:= TRUE;
			ELSE
				iInitStep 				:= 1000;		// Error step
			END_IF
		END_IF
	
	60: // Success - initialized flag, clear error
		bReInitialized					:= bInitialized;	// TRUE only when it's not first initialization e.g. online change
		bInitialized 					:= TRUE;
		bReInitializationError			:= FALSE;			// TRUE only when it's not first initialization e.g. online change
		bInitializationError			:= FALSE;
		iInitStep 						:= iInitStep + 10;
		
	70: // Idle
	
		;
		
	1000: // Error step
		wInitializationErrorCounter 	:= wInitializationErrorCounter + 1;
		IF wInitializationErrorCounter < 100 THEN
			iInitStep					:= iInitStep + 5;			// Go to delay
		ELSE
			bReInitializationError		:= bInitializationError;	// TRUE only when it's not first initialization e.g. online change
			bInitializationError		:= TRUE;
			bReInitialized				:= FALSE;
			iInitStep 					:= iInitStep + 10;
		END_IF

	1005: // Delay step
		tonDelay(IN:= TRUE, PT:= T#1S);
		IF tonDelay.Q THEN
			tonDelay(IN:= FALSE, PT:= T#1S);
			iInitStep					:= 0;
		END_IF
		
	1010: // Idle after error
		;
	
END_CASE

mcReadDriveAddress(	Axis				:= Axis,
					Execute				:= stMcAxisOnline.mcReadDriveAddress.bExecute,
					Done				=> stMcAxisOnline.mcReadDriveAddress.bDone,
					Busy				=> stMcAxisOnline.mcReadDriveAddress.bBusy,
					Error				=> stMcAxisOnline.mcReadDriveAddress.bError,
					ErrorID				=> stMcAxisOnline.mcReadDriveAddress.udiErrorID,
					DriveAddress		=> stMcAxisOnline.stDriveAddress);
				
mcReadParameterSet(	Parameter			:= stMcAxisOnline.stAxisParameter,
					Axis				:= Axis,
					Execute				:= stMcAxisOnline.mcReadParameterSet.bExecute,
					Done				=> stMcAxisOnline.mcReadParameterSet.bDone,
					Busy				=> stMcAxisOnline.mcReadParameterSet.bBusy,
					Error				=> stMcAxisOnline.mcReadParameterSet.bError,
					ErrorID				=> stMcAxisOnline.mcReadParameterSet.udiErrorID);
					
fbGetDriveRef(		bExecute			:= stMcAxisOnline.stGetDriveRef.bExecute,
					bBusy				=> stMcAxisOnline.stGetDriveRef.bBusy,
					bError				=> stMcAxisOnline.stGetDriveRef.bError,
					udiErrorID			=> stMcAxisOnline.stGetDriveRef.udiErrorID,
					stDriveRef			=> stMcAxisOnline.stDriveRef,
					Axis				:= Axis);
END_ACTION

ACTION ACT_Jog:
// Direct access from bSlow or bFast, if none then free choice
IF stMcAxisOnline.mcJog.bSlowForward OR stMcAxisOnline.mcJog.bSlowBackward THEN
	stMcAxisOnline.mcJog.eMode			:= MC_JOGMODE_STANDARD_SLOW;
ELSIF stMcAxisOnline.mcJog.bFastForward OR stMcAxisOnline.mcJog.bFastBackward THEN
	stMcAxisOnline.mcJog.eMode			:= MC_JOGMODE_STANDARD_FAST;
END_IF

mcJog(		Axis						:= Axis,
			JogForward					:= stMcAxisOnline.mcJog.bJogForward OR stMcAxisOnline.mcJog.bSlowForward OR stMcAxisOnline.mcJog.bFastForward,
			JogBackwards				:= stMcAxisOnline.mcJog.bJogBackwards OR stMcAxisOnline.mcJog.bSlowBackward OR stMcAxisOnline.mcJog.bFastBackward,
			Mode						:= stMcAxisOnline.mcJog.eMode,
			Position					:= stMcAxisOnline.mcJog.lrPosition,
			Velocity					:= stMcAxisOnline.mcJog.lrVelocity,
			Acceleration				:= stMcAxisOnline.mcJog.lrAcceleration,
			Deceleration				:= stMcAxisOnline.mcJog.lrDeceleration,
			Jerk						:= stMcAxisOnline.mcJog.lrJerk,
			Done						=> stMcAxisOnline.mcJog.bDone,
			Busy						=> stMcAxisOnline.mcJog.bBusy,
			Active						=> stMcAxisOnline.mcJog.bActive,
			CommandAborted				=> stMcAxisOnline.mcJog.bCommandAborted,
			Error						=> stMcAxisOnline.mcJog.bError,
			ErrorID						=> stMcAxisOnline.mcJog.udiErrorID);
END_ACTION

ACTION ACT_MotorMonitoring:
fbMotorMonitoring(	bReset				:= stMcAxisOnline.stMotorMonitoring.bReset,
					rTorqueLimit		:= stMcAxisOnline.stMotorMonitoring.rTorqueLimit,
					stDriveRef			:= stMcAxisOnline.stDriveRef,
					bError				=> stMcAxisOnline.stMotorMonitoring.bError,
					uiAdsErrId			=> stMcAxisOnline.stMotorMonitoring.uiAdsErrId,
					uiCANopenErrId		=> stMcAxisOnline.stMotorMonitoring.uiSecErrId,
					bInitialized		=> stMcAxisOnline.stMotorMonitoring.bInitialized,
					bWarning			=> stMcAxisOnline.stMotorMonitoring.bWarning,
					rWarningCurrent		=> stMcAxisOnline.stMotorMonitoring.rWarningCurrent,
					rTorquePerc			=> stMcAxisOnline.stMotorMonitoring.rTorquePerc,
					rTorquePercMax		=> stMcAxisOnline.stMotorMonitoring.rTorquePercMax,
					rTorque				=> stMcAxisOnline.stMotorMonitoring.rTorque,
					rTorqueF			=> stMcAxisOnline.stMotorMonitoring.rTorqueF,
					rTorqueMax			=> stMcAxisOnline.stMotorMonitoring.rTorqueMax,
					rCurrent			=> stMcAxisOnline.stMotorMonitoring.rCurrent,
					rCurrentF			=> stMcAxisOnline.stMotorMonitoring.rCurrentF,
					rCurrentMax			=> stMcAxisOnline.stMotorMonitoring.rCurrentMax,
					rI2T				=> stMcAxisOnline.stMotorMonitoring.rI2T,
					rI2TMax				=> stMcAxisOnline.stMotorMonitoring.rI2TMax,
					Axis				:= Axis);
END_ACTION

ACTION ACT_Move:
{region "Primary"}
mcMoveAbsolute(	Axis					:= Axis,
				Execute					:= stMcAxisOnline.mcMoveAbsolute.bExecute,
				Position				:= stMcAxisOnline.mcMoveAbsolute.lrPosition,
				Velocity				:= stMcAxisOnline.mcMoveAbsolute.lrVelocity,
				Acceleration			:= stMcAxisOnline.mcMoveAbsolute.lrAcceleration,
				Deceleration			:= stMcAxisOnline.mcMoveAbsolute.lrDeceleration,
				Jerk					:= stMcAxisOnline.mcMoveAbsolute.lrJerk,
				BufferMode				:= stMcAxisOnline.mcMoveAbsolute.eBufferMode,
				Options					:= stMcAxisOnline.mcMoveAbsolute.stOptions,
				Done					=> stMcAxisOnline.mcMoveAbsolute.bDone,
				Busy					=> stMcAxisOnline.mcMoveAbsolute.bBusy,
				Active					=> stMcAxisOnline.mcMoveAbsolute.bActive,
				CommandAborted			=> stMcAxisOnline.mcMoveAbsolute.bCommandAborted,
				Error					=> stMcAxisOnline.mcMoveAbsolute.bError,
				ErrorID					=> stMcAxisOnline.mcMoveAbsolute.udiErrorID);

mcMoveRelative(	Axis					:= Axis,
				Execute					:= stMcAxisOnline.mcMoveRelative.bExecute,
				Distance				:= stMcAxisOnline.mcMoveRelative.lrDistance,
				Velocity				:= stMcAxisOnline.mcMoveRelative.lrVelocity,
				Acceleration			:= stMcAxisOnline.mcMoveRelative.lrAcceleration,
				Deceleration			:= stMcAxisOnline.mcMoveRelative.lrDeceleration,
				Jerk					:= stMcAxisOnline.mcMoveRelative.lrJerk,
				BufferMode				:= stMcAxisOnline.mcMoveRelative.eBufferMode,
				Options					:= stMcAxisOnline.mcMoveRelative.stOptions,
				Done					=> stMcAxisOnline.mcMoveRelative.bDone,
				Busy					=> stMcAxisOnline.mcMoveRelative.bBusy,
				Active					=> stMcAxisOnline.mcMoveRelative.bActive,
				CommandAborted			=> stMcAxisOnline.mcMoveRelative.bCommandAborted,
				Error					=> stMcAxisOnline.mcMoveRelative.bError,
				ErrorID					=> stMcAxisOnline.mcMoveRelative.udiErrorID);
				
mcMoveVelocity(	Axis					:= Axis,
				Execute					:= stMcAxisOnline.mcMoveVelocity.bExecute,
				Velocity				:= stMcAxisOnline.mcMoveVelocity.lrVelocity,
				Acceleration			:= stMcAxisOnline.mcMoveVelocity.lrAcceleration,
				Deceleration			:= stMcAxisOnline.mcMoveVelocity.lrDeceleration,
				Jerk					:= stMcAxisOnline.mcMoveVelocity.lrJerk,
				Direction				:= stMcAxisOnline.mcMoveVelocity.eDirection,
				BufferMode				:= stMcAxisOnline.mcMoveVelocity.eBufferMode,
				Options					:= stMcAxisOnline.mcMoveVelocity.stOptions,
				InVelocity				=> stMcAxisOnline.mcMoveVelocity.bInVelocity,
				Busy					=> stMcAxisOnline.mcMoveVelocity.bBusy,
				Active					=> stMcAxisOnline.mcMoveVelocity.bActive,
				CommandAborted			=> stMcAxisOnline.mcMoveVelocity.bCommandAborted,
				Error					=> stMcAxisOnline.mcMoveVelocity.bError,
				ErrorID					=> stMcAxisOnline.mcMoveVelocity.udiErrorID);
stMcAxisOnline.mcMoveVelocity.bDone		:= stMcAxisOnline.mcMoveVelocity.bInVelocity;

mcMoveModulo(	Axis					:= Axis,
				Execute					:= stMcAxisOnline.mcMoveModulo.bExecute,
				Position				:= stMcAxisOnline.mcMoveModulo.lrPosition,
				Velocity				:= stMcAxisOnline.mcMoveModulo.lrVelocity,
				Acceleration			:= stMcAxisOnline.mcMoveModulo.lrAcceleration,
				Deceleration			:= stMcAxisOnline.mcMoveModulo.lrDeceleration,
				Jerk					:= stMcAxisOnline.mcMoveModulo.lrJerk,
				Direction				:= stMcAxisOnline.mcMoveModulo.eDirection,
				BufferMode				:= stMcAxisOnline.mcMoveModulo.eBufferMode,
				Options					:= stMcAxisOnline.mcMoveModulo.stOptions,
				Done					=> stMcAxisOnline.mcMoveModulo.bDone,
				Busy					=> stMcAxisOnline.mcMoveModulo.bBusy,
				Active					=> stMcAxisOnline.mcMoveModulo.bActive,
				CommandAborted			=> stMcAxisOnline.mcMoveModulo.bCommandAborted,
				Error					=> stMcAxisOnline.mcMoveModulo.bError,
				ErrorID					=> stMcAxisOnline.mcMoveModulo.udiErrorID);
{endregion}
{region "Secondary"}
mcMoveAbsolute2(Axis					:= Axis,
				Execute					:= stMcAxisOnline.mcMoveAbsolute2.bExecute,
				Position				:= stMcAxisOnline.mcMoveAbsolute2.lrPosition,
				Velocity				:= stMcAxisOnline.mcMoveAbsolute2.lrVelocity,
				Acceleration			:= stMcAxisOnline.mcMoveAbsolute2.lrAcceleration,
				Deceleration			:= stMcAxisOnline.mcMoveAbsolute2.lrDeceleration,
				Jerk					:= stMcAxisOnline.mcMoveAbsolute2.lrJerk,
				BufferMode				:= stMcAxisOnline.mcMoveAbsolute2.eBufferMode,
				Options					:= stMcAxisOnline.mcMoveAbsolute2.stOptions,
				Done					=> stMcAxisOnline.mcMoveAbsolute2.bDone,
				Busy					=> stMcAxisOnline.mcMoveAbsolute2.bBusy,
				Active					=> stMcAxisOnline.mcMoveAbsolute2.bActive,
				CommandAborted			=> stMcAxisOnline.mcMoveAbsolute2.bCommandAborted,
				Error					=> stMcAxisOnline.mcMoveAbsolute2.bError,
				ErrorID					=> stMcAxisOnline.mcMoveAbsolute2.udiErrorID);

mcMoveRelative2(Axis					:= Axis,
				Execute					:= stMcAxisOnline.mcMoveRelative2.bExecute,
				Distance				:= stMcAxisOnline.mcMoveRelative2.lrDistance,
				Velocity				:= stMcAxisOnline.mcMoveRelative2.lrVelocity,
				Acceleration			:= stMcAxisOnline.mcMoveRelative2.lrAcceleration,
				Deceleration			:= stMcAxisOnline.mcMoveRelative2.lrDeceleration,
				Jerk					:= stMcAxisOnline.mcMoveRelative2.lrJerk,
				BufferMode				:= stMcAxisOnline.mcMoveRelative2.eBufferMode,
				Options					:= stMcAxisOnline.mcMoveRelative2.stOptions,
				Done					=> stMcAxisOnline.mcMoveRelative2.bDone,
				Busy					=> stMcAxisOnline.mcMoveRelative2.bBusy,
				Active					=> stMcAxisOnline.mcMoveRelative2.bActive,
				CommandAborted			=> stMcAxisOnline.mcMoveRelative2.bCommandAborted,
				Error					=> stMcAxisOnline.mcMoveRelative2.bError,
				ErrorID					=> stMcAxisOnline.mcMoveRelative2.udiErrorID);
				
mcMoveVelocity2(Axis					:= Axis,
				Execute					:= stMcAxisOnline.mcMoveVelocity2.bExecute,
				Velocity				:= stMcAxisOnline.mcMoveVelocity2.lrVelocity,
				Acceleration			:= stMcAxisOnline.mcMoveVelocity2.lrAcceleration,
				Deceleration			:= stMcAxisOnline.mcMoveVelocity2.lrDeceleration,
				Jerk					:= stMcAxisOnline.mcMoveVelocity2.lrJerk,
				Direction				:= stMcAxisOnline.mcMoveVelocity2.eDirection,
				BufferMode				:= stMcAxisOnline.mcMoveVelocity2.eBufferMode,
				Options					:= stMcAxisOnline.mcMoveVelocity2.stOptions,
				InVelocity				=> stMcAxisOnline.mcMoveVelocity2.bInVelocity,
				Busy					=> stMcAxisOnline.mcMoveVelocity2.bBusy,
				Active					=> stMcAxisOnline.mcMoveVelocity2.bActive,
				CommandAborted			=> stMcAxisOnline.mcMoveVelocity2.bCommandAborted,
				Error					=> stMcAxisOnline.mcMoveVelocity2.bError,
				ErrorID					=> stMcAxisOnline.mcMoveVelocity2.udiErrorID);
stMcAxisOnline.mcMoveVelocity2.bDone	:= stMcAxisOnline.mcMoveVelocity2.bInVelocity;

mcMoveModulo2(	Axis					:= Axis,
				Execute					:= stMcAxisOnline.mcMoveModulo2.bExecute,
				Position				:= stMcAxisOnline.mcMoveModulo2.lrPosition,
				Velocity				:= stMcAxisOnline.mcMoveModulo2.lrVelocity,
				Acceleration			:= stMcAxisOnline.mcMoveModulo2.lrAcceleration,
				Deceleration			:= stMcAxisOnline.mcMoveModulo2.lrDeceleration,
				Jerk					:= stMcAxisOnline.mcMoveModulo2.lrJerk,
				Direction				:= stMcAxisOnline.mcMoveModulo2.eDirection,
				BufferMode				:= stMcAxisOnline.mcMoveModulo2.eBufferMode,
				Options					:= stMcAxisOnline.mcMoveModulo2.stOptions,
				Done					=> stMcAxisOnline.mcMoveModulo2.bDone,
				Busy					=> stMcAxisOnline.mcMoveModulo2.bBusy,
				Active					=> stMcAxisOnline.mcMoveModulo2.bActive,
				CommandAborted			=> stMcAxisOnline.mcMoveModulo2.bCommandAborted,
				Error					=> stMcAxisOnline.mcMoveModulo2.bError,
				ErrorID					=> stMcAxisOnline.mcMoveModulo2.udiErrorID);
{endregion}
END_ACTION

ACTION ACT_Power:
mcPower(	Axis						:= Axis,									//
			Enable						:= stMcAxisOnline.mcPower.bEnable,
			Enable_Positive				:= stMcAxisOnline.mcPower.bEnable_Positive,
			Enable_Negative				:= stMcAxisOnline.mcPower.bEnable_Negative,
			Override					:= stMcAxisOnline.mcPower.lrOverride,
			BufferMode					:= stMcAxisOnline.mcPower.eBufferMode,
			Options						:= stMcAxisOnline.mcPower.stOptions,
			Status						=> stMcAxisOnline.mcPower.bStatus,
			Busy						=> stMcAxisOnline.mcPower.bBusy,
			Active						=> stMcAxisOnline.mcPower.bActive,
			Error						=> stMcAxisOnline.mcPower.bError,
			ErrorID						=> stMcAxisOnline.mcPower.udiErrorID);
END_ACTION

ACTION ACT_Reset:
mcReset(	Axis						:= Axis,
			Execute						:= stMcAxisOnline.mcReset.bExecute,
			Done						=> stMcAxisOnline.mcReset.bDone,
			Busy						=> stMcAxisOnline.mcReset.bBusy,
			Error						=> stMcAxisOnline.mcReset.bError,
			ErrorID						=> stMcAxisOnline.mcReset.udiErrorID);
END_ACTION

ACTION ACT_SetPosition:
mcSetPosition(		Axis				:= Axis,
					Execute				:= stMcAxisOnline.mcSetPosition.bExecute,
					Position			:= stMcAxisOnline.mcSetPosition.lrPosition,
					Mode				:= stMcAxisOnline.mcSetPosition.bMode,
					Options				:= stMcAxisOnline.mcSetPosition.stOptions,
					Done				=> stMcAxisOnline.mcSetPosition.bDone,
					Busy				=> stMcAxisOnline.mcSetPosition.bBusy,
					Error				=> stMcAxisOnline.mcSetPosition.bError,
					ErrorID				=> stMcAxisOnline.mcSetPosition.udiErrorID);
END_ACTION

ACTION ACT_SetPositionIO:

;(*fbSetPositionOffset(Execute				:= stMcAxisOnline.stSetPositionOffset.bExecute,
					Position			:= stMcAxisOnline.stSetPositionOffset.lrPosition,
					Relative			:= stMcAxisOnline.stSetPositionOffset.bRelative,
					Feedback			:= stMcAxisOnline.stSetPositionOffset.eFeedback,
					Memory				:= stMcAxisOnline.stSetPositionOffset.eMemory,
					Busy				=> stMcAxisOnline.stSetPositionOffset.bBusy,
					Error				=> stMcAxisOnline.stSetPositionOffset.bError,
					ErrorID				=> stMcAxisOnline.stSetPositionOffset.udiErrorID,
					Axis				:= Axis);
					*)
END_ACTION

ACTION ACT_States:
// Read States and forward main states
Axis.ReadStatus();
stMcAxisOnline.stStatus.stAxisStatus		:= Axis.Status;
stMcAxisOnline.stStatus.dwAxisId			:= Axis.NcToPlc.AxisId;
stMcAxisOnline.stStatus.bNcError			:= Axis.Status.Error;
stMcAxisOnline.stStatus.udiNcErrorCode		:= Axis.Status.ErrorID;
stMcAxisOnline.stStatus.udiNcErrorCodeHex	:= Axis.Status.ErrorID;

stMcAxisOnline.stStatus.sAxisName			:= stMcAxisOnline.stAxisParameter.sAxisName;
stMcAxisOnline.stStatus.lrActPos			:= Axis.NcToPlc.ActPos;
stMcAxisOnline.stStatus.lrModuloActPos		:= Axis.NcToPlc.ModuloActPos;
stMcAxisOnline.stStatus.lrActVelo			:= Axis.NcToPlc.ActVelo;
stMcAxisOnline.stStatus.lrActAcc			:= Axis.NcToPlc.ActAcc;
stMcAxisOnline.stStatus.lrActTorque			:= Axis.NcToPlc.ActTorque;
stMcAxisOnline.stStatus.lrPosDiff			:= Axis.NcToPlc.PosDiff;
stMcAxisOnline.stStatus.lrSetPos			:= Axis.NcToPlc.SetPos;
stMcAxisOnline.stStatus.lrSetVelo			:= Axis.NcToPlc.SetVelo;
stMcAxisOnline.stStatus.lrSetAcc			:= Axis.NcToPlc.SetAcc;
stMcAxisOnline.stStatus.lrSetTorque			:= Axis.NcToPlc.SetTorque;
stMcAxisOnline.stStatus.lrPosDiff			:= Axis.NcToPlc.PosDiff;
stMcAxisOnline.stStatus.bAxisReady			:= Axis.Status.Operational;
stMcAxisOnline.stStatus.bHomed				:= Axis.Status.Homed;
stMcAxisOnline.stStatus.bCoupled			:= Axis.Status.Coupled;

// zezwolenie na zjazd z krancowki hw
Axis.PlcToNc.ControlDWord.8				:= stMcAxisOnline.stStatus.bAcceptBlockedDrive;
END_ACTION

ACTION ACT_Stop:
mcHalt(		Axis						:= Axis,
			Execute						:= stMcAxisOnline.mcHalt.bExecute,
			Deceleration				:= stMcAxisOnline.mcHalt.lrDeceleration,
			Jerk						:= stMcAxisOnline.mcHalt.lrJerk,
			BufferMode					:= stMcAxisOnline.mcHalt.eBufferMode,
			Options						:= stMcAxisOnline.mcHalt.stOptions,
			Done						=> stMcAxisOnline.mcHalt.bDone,
			Busy						=> stMcAxisOnline.mcHalt.bBusy,
			Active						=> stMcAxisOnline.mcHalt.bActive,
			CommandAborted				=> stMcAxisOnline.mcHalt.bCommandAborted,
			Error						=> stMcAxisOnline.mcHalt.bError,
			ErrorID						=> stMcAxisOnline.mcHalt.udiErrorID);
			
mcStop(		Axis						:= Axis,
			Execute						:= stMcAxisOnline.mcStop.bExecute,
			Deceleration				:= stMcAxisOnline.mcStop.lrDeceleration,
			Jerk						:= stMcAxisOnline.mcStop.lrJerk,
			Options						:= stMcAxisOnline.mcStop.stOptions,
			Done						=> stMcAxisOnline.mcStop.bDone,
			Busy						=> stMcAxisOnline.mcStop.bBusy,
			Active						=> stMcAxisOnline.mcStop.bActive,
			CommandAborted				=> stMcAxisOnline.mcStop.bCommandAborted,
			Error						=> stMcAxisOnline.mcStop.bError,
			ErrorID						=> stMcAxisOnline.mcStop.udiErrorID);
			
mcStopSS2(	Axis						:= Axis,
			Execute						:= stMcAxisOnline.mcSS2.bExecute,
			Deceleration				:= stMcAxisOnline.mcSS2.lrDeceleration,
			Jerk						:= stMcAxisOnline.mcSS2.lrJerk,
			Options						:= stMcAxisOnline.mcSS2.stOptions,
			Done						=> stMcAxisOnline.mcSS2.bDone,
			Busy						=> stMcAxisOnline.mcSS2.bBusy,
			Active						=> stMcAxisOnline.mcSS2.bActive,
			CommandAborted				=> stMcAxisOnline.mcSS2.bCommandAborted,
			Error						=> stMcAxisOnline.mcSS2.bError,
			ErrorID						=> stMcAxisOnline.mcSS2.udiErrorID);
			
mcStopSS1(	Axis						:= Axis,
			Execute						:= stMcAxisOnline.mcSS1.bExecute,
			Deceleration				:= stMcAxisOnline.mcSS1.lrDeceleration,
			Jerk						:= stMcAxisOnline.mcSS1.lrJerk,
			Options						:= stMcAxisOnline.mcSS1.stOptions,
			Done						=> stMcAxisOnline.mcSS1.bDone,
			Busy						=> stMcAxisOnline.mcSS1.bBusy,
			Active						=> stMcAxisOnline.mcSS1.bActive,
			CommandAborted				=> stMcAxisOnline.mcSS1.bCommandAborted,
			Error						=> stMcAxisOnline.mcSS1.bError,
			ErrorID						=> stMcAxisOnline.mcSS1.udiErrorID);
// SS1 - after MC_Stop function we have to disable drive			
stMcAxisOnline.mcPower.bEnable R= stMcAxisOnline.mcPower.bEnable_Positive R= stMcAxisOnline.mcPower.bEnable_Negative R= (stMcAxisOnline.mcSS1.bDone OR stMcAxisOnline.mcSS1.bCommandAborted OR stMcAxisOnline.mcSS1.bError);
END_ACTION

ACTION ACT_SWLimitSwitch:
fbNcLimitSwitch(	udiAxisID		:= Axis.NcToPlc.AxisId, 
					bRead			:= stMcAxisOnline.stNcLimitSwitch.bRead, 
					bWrite			:= stMcAxisOnline.stNcLimitSwitch.bWrite, 
					bReset			:= stMcAxisOnline.stNcLimitSwitch.bReset, 
					lrSetMinPos		:= stMcAxisOnline.stNcLimitSwitch.lrSetMinPos, 
					lrSetMaxPos		:= stMcAxisOnline.stNcLimitSwitch.lrSetMaxPos, 
					bSetMinMon		:= stMcAxisOnline.stNcLimitSwitch.bSetMinMon, 
					bSetMaxMon		:= stMcAxisOnline.stNcLimitSwitch.bSetMaxMon, 
					bBusy			=> stMcAxisOnline.stNcLimitSwitch.bBusy, 
					bError			=> stMcAxisOnline.stNcLimitSwitch.bError, 
					udiErrorID		=> stMcAxisOnline.stNcLimitSwitch.udiErrorID, 
					lrActMinPos		=> stMcAxisOnline.stNcLimitSwitch.lrActMinPos, 
					lrActMaxPos		=> stMcAxisOnline.stNcLimitSwitch.lrActMaxPos, 
					bActMinMon		=> stMcAxisOnline.stNcLimitSwitch.bActMinMon, 
					bActMaxMon		=> stMcAxisOnline.stNcLimitSwitch.bActMaxMon);
END_ACTION

END_FUNCTION_BLOCK

// ---- POUs/FB/POUsAxisOnline/EL72xx/FB_MotorMonitoringEL72xx.TcPOU
//==================================================================================================
//							Beckhoff Automation Poland
//									9.07.2018
//	Blok funkcyjny pozwala na monitorowanie i ograniczanie momentu oraz monitoring parametru I2T dla EL72xx.
//	Zmienne do zlinkowania zadeklarowane są wewnątrz bloku.
//	Ograniczenie i monitorowanie momentu
//	Ograniczenie momentu podawane jest przez wejście rTorqueLimit.
//	Na wyjściu podana jest wartość surowa w %, jak i przeskalowana na A (prąd) i Nm (moment).
//	Blok zwraca wartości bieżące, przefiltrowane i maksymalne.
//	Wartości maksymalne mogą być wyzerowane za pomocą zmiennej bReset.
//	Wewnętrznie wykorzystany jest blok FB_FilterEx.
//
//  v1.0	|| TC v 3.1.4022.22		|| - pierwsza wersja
//==================================================================================================
FUNCTION_BLOCK FB_MotorMonitoringEL72xx
VAR CONSTANT
	rTorqueLimitLow					: REAL 		:= 0.01;				// Low limit used for bipolar torque limit value
	rTorqueLimitHigh				: REAL		:= 500.0;				// High limit used for bipolar torque limit value
END_VAR
VAR_INPUT
	bReset							: BOOL;								// Reset FB
	rTorqueLimit					: REAL 		:= rTorqueLimitHigh; 	// Bipolar torque limit: 0-500%, resolution 0.1%, value goes to: 16#6072 (Ch A)/ 16#6872 (Ch B)	
	stDriveRef						: ST_DriveRef;						// Necessary for FB_CoERead_ByDriveRef
END_VAR
VAR_OUTPUT
	bError							: BOOL; 							// General error: parameter or CoE read.
																		// If bError = TRUE and bInitialized = FALSE - error during read motor data.
																		// If bError = TRUE and bInitialized = TRUE and (iAdsErrId <> 0 or iCANopenErrId <> 0) then I2T read error
																		// If bError = TRUE and bInitialized = TRUE and iAdsErrId = 0 and iCANopenErrId = 0 then parameter error: rTorqueLimit outside permitted range rTorqueLimitLow..rTorqueLimitHigh or Empty stDriveRef
	uiAdsErrId						: UINT;								// Forwarded output FB_CoERead_ByDriveRef
	uiCANopenErrId					: UINT;								// Forwarded output FB_CoERead_ByDriveRef
	bInitialized					: BOOL;								// TRUE - Motor data read without errors, so it's possible to calculate torqe and current values in metric units
	bWarning						: BOOL;								// rCurrentF > rWarningCurrent, be aware to be over permitted range
	rWarningCurrent					: REAL; 							// 8011:12 - Rated current in [A]
	rTorquePerc						: REAL;								// [%]
	rTorquePercMax					: REAL;								// Max [%]
	rTorque							: REAL; 							// [Nm]
	rTorqueF						: REAL;								// Filtered [Nm]
	rTorqueMax						: REAL;								// Max [Nm]
	rCurrent						: REAL; 							// [A]
	rCurrentF						: REAL;								// Filtered [A]
	rCurrentMax						: REAL;								// Max [A]
	rI2T							: REAL; 							// Thermal Motor Utilization: 16#32C1:02 (Ch A)/ 16#36C1:02 (Ch B); units: [%]
	rI2TMax							: REAL; 							// Max % Nominal
END_VAR
VAR_IN_OUT
	Axis							: AXIS_REF;							// Axis Ref struct
END_VAR
VAR
//======================= Internal var ===========================
	iStep							: INT;								// Case instruction
	bDriveRefOK						: BOOL;								// stDriveRef contains necessary data to read CoE
	bTorqueLimitOK					: BOOL;								// rTorqueLimit in permitted range rTorqueLimitLow..rTorqueLimitHigh
	uiBipolarTorqueLimitValue  		AT %Q*: UINT; 						// Raw data, linked to Bipolar torque limit value
	rTorqueRAW						: REAL; 							// -1000 .. 1000 - RAW values the same as process image
	rSfTorque						: REAL; 							// A --> Nm
	rSfCurrent						: REAL; 							// RAW -1000..1000 --> A
	wInitErrorCount					: WORD;								// Initialization error counter, if bigger then 10 then error
	rPeakCurrent					: REAL; 							// 8011:11 in [A]
	rRatedCurrent					: REAL; 							// 8011:12 in [A]
	bFirstCycle						: BOOL := TRUE;
	bRMSValue						: BOOL;								// 16#8010:54  Bit 0 = 1 - RMS value
//========================== EL72xx =============================
	dwPeakCurrent					: DWORD;							// 16#8011:11 - Max current, Peak current [mA]
	dwRatedCurrent					: DWORD;							// 16#8011:12 - Rated current [mA]
	dwTorqueConstant				: DWORD;							// 16#8011:16 - Torque constant [mNm/A]
	dwFeatureBits					: DWORD;							// 16#8010:54 - Feature bits:	Peak value --> Bit 0 = 0 (default for EL7201-000x) 
																									//	RMS value --> Bit 0 = 1 (default for EL7211-000x)
//========================== I2T ================================
	sDeviceName						: STRING;							// 
	sNo								: STRING(1);						// xxxxxxx-000Y - char Y
	usiI2T							: USINT;							// 
	bDS402Profile					: BOOL;								// Flag DS402
	bMDP742Profile					: BOOL;								// Flag MDP742
	wMotorI2TIndex					: WORD;								// EL72x1-0000 --> MDP 742: A011:11 Motor I2T temperature [%] USINT
																		// EL72x1-0001 --> DS 402: 2031:11 Motor I2T temperature [%] USINT
//========================== FBs ================================
	rtReset							: R_TRIG;							// Reset trigger
	tonWait							: TON;								// Wait timer
	fbFilterEx						: FB_FilterEx;						// Filter
	fbGETCURTASKINDEX   			: GETCURTASKINDEX;					// FB to check task no
	fbCoERead						: FB_CoERead_ByDriveRef;			// FB for read CoE parameters
//===============================================================
END_VAR

